(* CODESYS project IOoverNode

Project tree, tasks and I/O mapping:
  Device : XC303, Eaton Automation, version 3.5.16.60
      unmapped channels: Output, Input
    application Application
      libraries: EA_XN300_CAN, 3.5.7.3 (Eaton Automation); Standard, 3.5.15.0 (System); CAA CiA 405, 3.5.15.0 (CAA Technical Workgroup)
      task DatasourcesTask (cyclic, interval 50 ms, priority 31) calls Datasources.Datasources_PRG
      task MainTask (cyclic, interval t#10ms, priority 1) calls PLC_PRG
      function block InputData [ST]
      program PLC_PRG [ST]
      program PRG_PLC [CFC]
    CANbus : CANbus, Eaton Automation, order no. 
      , version 3.5.15.0
        settings: Baudrate = 500 kbit/s
      CANopen_Manager : CANopen_Manager, Eaton Automation, version 3.5.16.0
          settings: CANopen NodeID = 10; ConfigVersion = 50659584
        DA1 : DA1, Eaton Industries, order no. 0, version 3.5.16.100
            settings: General Options.Optional Device = TRUE; NODEIDSAVED = 4; SDO Timeout = 1000000; PDO_Autoconfig = FALSE; EXPERTSETTINGS = True; Emergency-General Parameters.Emergency COBID = 16#00000084; Heartbeat-Producer Time = 200; PDO 16#1400.COBID = 16#40000204; Process by CANopenManager = TRUE; PDO 16#1401.COBID = 16#C0000304; Generic COBID = '$NODEID+16#C0000300'; Process by CANopenManager = TRUE; PDO 16#1800.COBID = 16#40000184; PDO 16#1800.Transmission Type = 16#FF; PDO 16#1800.Event Timer = 0; Process by CANopenManager = TRUE; PDO 16#1801.COBID = 16#C0000284; PDO 16#1801.Event Timer = 0; Generic COBID = '$NODEID+16#C0000280'; Process by CANopenManager = TRUE; Control Command Register.Subindex = 16#00; Speed Reference.Subindex = 16#00; Torque Reference.Subindex = 16#00; User Ramp.Subindex = 16#00; no-name.Index = 16#0006; no-name.Subindex = 16#00; no-name.Index = 16#0006; no-name.Subindex = 16#00; no-name.Index = 16#0006; no-name.Subindex = 16#00; no-name.Index = 16#0006; no-name.Subindex = 16#00; Drive Status Register.Subindex = 16#00; Motor Speed.Subindex = 16#00; Motor Current.Subindex = 16#00; Motor Torque.Subindex = 16#00; Motor Power.Subindex = 16#00; Drive Temperature.Subindex = 16#00; DC Bus Voltage.Subindex = 16#00; Motor Speed (Internal).Subindex = 16#00;
              SDO List.Set COB-ID sync.Index = 16#1005; SDO List.Set COB-ID sync.Subindex = 16#00; SDO List.Set COB-ID sync.Value = 16#00000080; SDO List.Set COB-ID sync.Size = 32; SDO List.Set COB-ID sync.AbortIfError = FALSE; SDO List.Set COB-ID sync.JumpToLine = FALSE; SDO List.Set COB-ID sync.Line = 0; SDO List.Set Guardtime.Index = 16#100C; SDO List.Set Guardtime.Subindex = 16#00; SDO List.Set Guardtime.Value = 16#00000000; SDO List.Set Guardtime.Size = 16; SDO List.Set Guardtime.AbortIfError = FALSE; SDO List.Set Guardtime.JumpToLine = FALSE; SDO List.Set Guardtime.Line = 0; SDO List.Set Lifetime.Index = 16#100D; SDO List.Set Lifetime.Subindex = 16#00; SDO List.Set Lifetime.Value = 16#00000000; SDO List.Set Lifetime.Size = 8; SDO List.Set Lifetime.AbortIfError = FALSE; SDO List.Set Lifetime.JumpToLine = FALSE; SDO List.Set Lifetime.Line = 0; SDO List.Disable Emcy CobID.Index = 16#1014; SDO List.Disable Emcy CobID.Subindex = 16#00; SDO List.Disable Emcy CobID.Value = 16#80000084; SDO List.Disable Emcy CobID.Size = 32; SDO List.Disable Emcy CobID.AbortIfError = FALSE; SDO List.Disable Emcy CobID.JumpToLine = FALSE; SDO List.Disable Emcy CobID.Line = 0; SDO List.Set Emcy CobID.Index = 16#1014; SDO List.Set Emcy CobID.Subindex = 16#00; SDO List.Set Emcy CobID.Value = 16#00000084; SDO List.Set Emcy CobID.Size = 32; SDO List.Set Emcy CobID.AbortIfError = FALSE; SDO List.Set Emcy CobID.JumpToLine = FALSE; SDO List.Set Emcy CobID.Line = 0; SDO List.Set Heartbeat Producer.Index = 16#1017; SDO List.Set Heartbeat Producer.Subindex = 16#00; SDO List.Set Heartbeat Producer.Value = 16#000000C8; SDO List.Set Heartbeat Producer.Size = 16; SDO List.Set Heartbeat Producer.AbortIfError = FALSE;
              SDO List.Set Heartbeat Producer.JumpToLine = FALSE; SDO List.Set Heartbeat Producer.Line = 0; SDO List.Disable PDO.Index = 16#1400; SDO List.Disable PDO.Subindex = 16#01; SDO List.Disable PDO.Value = 16#C0000204; SDO List.Disable PDO.Size = 32; SDO List.Disable PDO.AbortIfError = FALSE; SDO List.Disable PDO.JumpToLine = FALSE; SDO List.Disable PDO.Line = 0; SDO List.Set transmission type.Index = 16#1400; SDO List.Set transmission type.Subindex = 16#02; SDO List.Set transmission type.Value = 16#FE; SDO List.Set transmission type.Size = 8; SDO List.Set transmission type.AbortIfError = FALSE; SDO List.Set transmission type.JumpToLine = FALSE; SDO List.Set transmission type.Line = 0; SDO List.Clear pdo mapping.Index = 16#1600; SDO List.Clear pdo mapping.Subindex = 16#00; SDO List.Clear pdo mapping.Value = 16#0; SDO List.Clear pdo mapping.Size = 8; SDO List.Clear pdo mapping.AbortIfError = FALSE; SDO List.Clear pdo mapping.JumpToLine = FALSE; SDO List.Clear pdo mapping.Line = 0; SDO List.Set Mapping.Index = 16#1600; SDO List.Set Mapping.Subindex = 16#01; SDO List.Set Mapping.Value = 16#20000010; SDO List.Set Mapping.Size = 32; SDO List.Set Mapping.AbortIfError = FALSE; SDO List.Set Mapping.JumpToLine = FALSE; SDO List.Set Mapping.Line = 0; SDO List.Set Mapping.Index = 16#1600; SDO List.Set Mapping.Subindex = 16#02; SDO List.Set Mapping.Value = 16#20010010; SDO List.Set Mapping.Size = 32; SDO List.Set Mapping.AbortIfError = FALSE; SDO List.Set Mapping.JumpToLine = FALSE; SDO List.Set Mapping.Line = 0; SDO List.Set Mapping.Index = 16#1600; SDO List.Set Mapping.Subindex = 16#03; SDO List.Set Mapping.Value = 16#20020010;
              SDO List.Set Mapping.Size = 32; SDO List.Set Mapping.AbortIfError = FALSE; SDO List.Set Mapping.JumpToLine = FALSE; SDO List.Set Mapping.Line = 0; SDO List.Set Mapping.Index = 16#1600; SDO List.Set Mapping.Subindex = 16#04; SDO List.Set Mapping.Value = 16#20030010; SDO List.Set Mapping.Size = 32; SDO List.Set Mapping.AbortIfError = FALSE; SDO List.Set Mapping.JumpToLine = FALSE; SDO List.Set Mapping.Line = 0; SDO List.Set number of mappings.Index = 16#1600; SDO List.Set number of mappings.Subindex = 16#00; SDO List.Set number of mappings.Value = 16#04; SDO List.Set number of mappings.Size = 8; SDO List.Set number of mappings.AbortIfError = FALSE; SDO List.Set number of mappings.JumpToLine = FALSE; SDO List.Set number of mappings.Line = 0; SDO List.Set and enable COB-ID.Index = 16#1400; SDO List.Set and enable COB-ID.Subindex = 16#01; SDO List.Set and enable COB-ID.Value = 16#40000204; SDO List.Set and enable COB-ID.Size = 32; SDO List.Set and enable COB-ID.AbortIfError = FALSE; SDO List.Set and enable COB-ID.JumpToLine = FALSE; SDO List.Set and enable COB-ID.Line = 0; SDO List.Disable PDO.Index = 16#1401; SDO List.Disable PDO.Subindex = 16#01; SDO List.Disable PDO.Value = 16#C0000304; SDO List.Disable PDO.Size = 32; SDO List.Disable PDO.AbortIfError = FALSE; SDO List.Disable PDO.JumpToLine = FALSE; SDO List.Disable PDO.Line = 0; SDO List.Disable PDO.Index = 16#1800; SDO List.Disable PDO.Subindex = 16#01; SDO List.Disable PDO.Value = 16#C0000184; SDO List.Disable PDO.Size = 32; SDO List.Disable PDO.AbortIfError = FALSE; SDO List.Disable PDO.JumpToLine = FALSE; SDO List.Disable PDO.Line = 0; SDO List.Set transmission type.Index = 16#1800;
              SDO List.Set transmission type.Subindex = 16#02; SDO List.Set transmission type.Value = 16#FF; SDO List.Set transmission type.Size = 8; SDO List.Set transmission type.AbortIfError = FALSE; SDO List.Set transmission type.JumpToLine = FALSE; SDO List.Set transmission type.Line = 0; SDO List.Set inhibit time.Index = 16#1800; SDO List.Set inhibit time.Subindex = 16#03; SDO List.Set inhibit time.Value = 16#0000; SDO List.Set inhibit time.Size = 16; SDO List.Set inhibit time.AbortIfError = FALSE; SDO List.Set inhibit time.JumpToLine = FALSE; SDO List.Set inhibit time.Line = 0; SDO List.Clear pdo mapping.Index = 16#1A00; SDO List.Clear pdo mapping.Subindex = 16#00; SDO List.Clear pdo mapping.Value = 16#0; SDO List.Clear pdo mapping.Size = 8; SDO List.Clear pdo mapping.AbortIfError = FALSE; SDO List.Clear pdo mapping.JumpToLine = FALSE; SDO List.Clear pdo mapping.Line = 0; SDO List.Set Mapping.Index = 16#1A00; SDO List.Set Mapping.Subindex = 16#01; SDO List.Set Mapping.Value = 16#200A0010; SDO List.Set Mapping.Size = 32; SDO List.Set Mapping.AbortIfError = FALSE; SDO List.Set Mapping.JumpToLine = FALSE; SDO List.Set Mapping.Line = 0; SDO List.Set Mapping.Index = 16#1A00; SDO List.Set Mapping.Subindex = 16#02; SDO List.Set Mapping.Value = 16#200B0010; SDO List.Set Mapping.Size = 32; SDO List.Set Mapping.AbortIfError = FALSE; SDO List.Set Mapping.JumpToLine = FALSE; SDO List.Set Mapping.Line = 0; SDO List.Set Mapping.Index = 16#1A00; SDO List.Set Mapping.Subindex = 16#03; SDO List.Set Mapping.Value = 16#200D0010; SDO List.Set Mapping.Size = 32; SDO List.Set Mapping.AbortIfError = FALSE; SDO List.Set Mapping.JumpToLine = FALSE;
              SDO List.Set Mapping.Line = 0; SDO List.Set Mapping.Index = 16#1A00; SDO List.Set Mapping.Subindex = 16#04; SDO List.Set Mapping.Value = 16#200E0010; SDO List.Set Mapping.Size = 32; SDO List.Set Mapping.AbortIfError = FALSE; SDO List.Set Mapping.JumpToLine = FALSE; SDO List.Set Mapping.Line = 0; SDO List.Set number of mappings.Index = 16#1A00; SDO List.Set number of mappings.Subindex = 16#00; SDO List.Set number of mappings.Value = 16#04; SDO List.Set number of mappings.Size = 8; SDO List.Set number of mappings.AbortIfError = FALSE; SDO List.Set number of mappings.JumpToLine = FALSE; SDO List.Set number of mappings.Line = 0; SDO List.Set and enable COB-ID.Index = 16#1800; SDO List.Set and enable COB-ID.Subindex = 16#01; SDO List.Set and enable COB-ID.Value = 16#40000184; SDO List.Set and enable COB-ID.Size = 32; SDO List.Set and enable COB-ID.AbortIfError = FALSE; SDO List.Set and enable COB-ID.JumpToLine = FALSE; SDO List.Set and enable COB-ID.Line = 0; SDO List.Disable PDO.Index = 16#1801; SDO List.Disable PDO.Subindex = 16#01; SDO List.Disable PDO.Value = 16#C0000284; SDO List.Disable PDO.Size = 32; SDO List.Disable PDO.AbortIfError = FALSE; SDO List.Disable PDO.JumpToLine = FALSE; SDO List.Disable PDO.Line = 0; ConfigVersion = 50659584
            unmapped channels: Control Command Register, Speed Reference, Torque Reference, User Ramp, Drive Status Register, Motor Speed, Motor Current, Motor Torque
        DC1 : DC1, Eaton, order no. 0, version 3.5.16.100
            settings: General Options.Optional Device = TRUE; NODEIDSAVED = 3; SDO Timeout = 1000000; PDO_Autoconfig = FALSE; EXPERTSETTINGS = True; Emergency-General Parameters.Emergency COBID = 16#00000083; Heartbeat-Producer Time = 200; PDO 16#1400.COBID = 16#40000203; PDO 16#1400.Transmission Type = 16#FE; Process by CANopenManager = TRUE; PDO 16#1401.COBID = 16#C0000303; Generic COBID = '$NODEID+16#C0000300'; Process by CANopenManager = TRUE; PDO 16#1800.COBID = 16#40000183; PDO 16#1800.Event Timer = 0; Process by CANopenManager = TRUE; PDO 16#1801.COBID = 16#C0000283; PDO 16#1801.Event Timer = 0; Generic COBID = '$NODEID+16#C0000280'; Process by CANopenManager = TRUE; Control Command Register.Subindex = 16#00; Speed Reference.Subindex = 16#00; User Ramp.Subindex = 16#00; no-name.Index = 16#0006; no-name.Subindex = 16#00; no-name.Index = 16#0006; no-name.Subindex = 16#00; no-name.Index = 16#0006; no-name.Subindex = 16#00; no-name.Index = 16#0006; no-name.Subindex = 16#00; Drive Status Register.Subindex = 16#00; Motor Speed.Subindex = 16#00; Motor Current.Subindex = 16#00; Drive Temperature.Subindex = 16#00; DC Bus Voltage.Subindex = 16#00; Digital Input Status.Subindex = 16#00; Analog Input 1.Subindex = 16#00; Analog Input 2.Subindex = 16#00; SDO List.Set COB-ID sync.Index = 16#1005;
              SDO List.Set COB-ID sync.Subindex = 16#00; SDO List.Set COB-ID sync.Value = 16#00000080; SDO List.Set COB-ID sync.Size = 32; SDO List.Set COB-ID sync.AbortIfError = FALSE; SDO List.Set COB-ID sync.JumpToLine = FALSE; SDO List.Set COB-ID sync.Line = 0; SDO List.Set Guardtime.Index = 16#100C; SDO List.Set Guardtime.Subindex = 16#00; SDO List.Set Guardtime.Value = 16#00000000; SDO List.Set Guardtime.Size = 16; SDO List.Set Guardtime.AbortIfError = FALSE; SDO List.Set Guardtime.JumpToLine = FALSE; SDO List.Set Guardtime.Line = 0; SDO List.Set Lifetime.Index = 16#100D; SDO List.Set Lifetime.Subindex = 16#00; SDO List.Set Lifetime.Value = 16#00000000; SDO List.Set Lifetime.Size = 8; SDO List.Set Lifetime.AbortIfError = FALSE; SDO List.Set Lifetime.JumpToLine = FALSE; SDO List.Set Lifetime.Line = 0; SDO List.Disable Emcy CobID.Index = 16#1014; SDO List.Disable Emcy CobID.Subindex = 16#00; SDO List.Disable Emcy CobID.Value = 16#80000083; SDO List.Disable Emcy CobID.Size = 32; SDO List.Disable Emcy CobID.AbortIfError = FALSE; SDO List.Disable Emcy CobID.JumpToLine = FALSE; SDO List.Disable Emcy CobID.Line = 0; SDO List.Set Emcy CobID.Index = 16#1014; SDO List.Set Emcy CobID.Subindex = 16#00; SDO List.Set Emcy CobID.Value = 16#00000083; SDO List.Set Emcy CobID.Size = 32; SDO List.Set Emcy CobID.AbortIfError = FALSE; SDO List.Set Emcy CobID.JumpToLine = FALSE; SDO List.Set Emcy CobID.Line = 0; SDO List.Set Heartbeat Producer.Index = 16#1017; SDO List.Set Heartbeat Producer.Subindex = 16#00; SDO List.Set Heartbeat Producer.Value = 16#000000C8; SDO List.Set Heartbeat Producer.Size = 16; SDO List.Set Heartbeat Producer.AbortIfError = FALSE; SDO List.Set Heartbeat Producer.JumpToLine = FALSE;
              SDO List.Set Heartbeat Producer.Line = 0; SDO List.Disable PDO.Index = 16#1400; SDO List.Disable PDO.Subindex = 16#01; SDO List.Disable PDO.Value = 16#C0000203; SDO List.Disable PDO.Size = 32; SDO List.Disable PDO.AbortIfError = FALSE; SDO List.Disable PDO.JumpToLine = FALSE; SDO List.Disable PDO.Line = 0; SDO List.Set transmission type.Index = 16#1400; SDO List.Set transmission type.Subindex = 16#02; SDO List.Set transmission type.Value = 16#FE; SDO List.Set transmission type.Size = 8; SDO List.Set transmission type.AbortIfError = FALSE; SDO List.Set transmission type.JumpToLine = FALSE; SDO List.Set transmission type.Line = 0; SDO List.Clear pdo mapping.Index = 16#1600; SDO List.Clear pdo mapping.Subindex = 16#00; SDO List.Clear pdo mapping.Value = 16#0; SDO List.Clear pdo mapping.Size = 8; SDO List.Clear pdo mapping.AbortIfError = FALSE; SDO List.Clear pdo mapping.JumpToLine = FALSE; SDO List.Clear pdo mapping.Line = 0; SDO List.Set Mapping.Index = 16#1600; SDO List.Set Mapping.Subindex = 16#01; SDO List.Set Mapping.Value = 16#20000010; SDO List.Set Mapping.Size = 32; SDO List.Set Mapping.AbortIfError = FALSE; SDO List.Set Mapping.JumpToLine = FALSE; SDO List.Set Mapping.Line = 0; SDO List.Set Mapping.Index = 16#1600; SDO List.Set Mapping.Subindex = 16#02; SDO List.Set Mapping.Value = 16#20010010; SDO List.Set Mapping.Size = 32; SDO List.Set Mapping.AbortIfError = FALSE; SDO List.Set Mapping.JumpToLine = FALSE; SDO List.Set Mapping.Line = 0; SDO List.Set Mapping.Index = 16#1600; SDO List.Set Mapping.Subindex = 16#03; SDO List.Set Mapping.Value = 16#20030010; SDO List.Set Mapping.Size = 32;
              SDO List.Set Mapping.AbortIfError = FALSE; SDO List.Set Mapping.JumpToLine = FALSE; SDO List.Set Mapping.Line = 0; SDO List.Set number of mappings.Index = 16#1600; SDO List.Set number of mappings.Subindex = 16#00; SDO List.Set number of mappings.Value = 16#03; SDO List.Set number of mappings.Size = 8; SDO List.Set number of mappings.AbortIfError = FALSE; SDO List.Set number of mappings.JumpToLine = FALSE; SDO List.Set number of mappings.Line = 0; SDO List.Set and enable COB-ID.Index = 16#1400; SDO List.Set and enable COB-ID.Subindex = 16#01; SDO List.Set and enable COB-ID.Value = 16#40000203; SDO List.Set and enable COB-ID.Size = 32; SDO List.Set and enable COB-ID.AbortIfError = FALSE; SDO List.Set and enable COB-ID.JumpToLine = FALSE; SDO List.Set and enable COB-ID.Line = 0; SDO List.Disable PDO.Index = 16#1401; SDO List.Disable PDO.Subindex = 16#01; SDO List.Disable PDO.Value = 16#C0000303; SDO List.Disable PDO.Size = 32; SDO List.Disable PDO.AbortIfError = FALSE; SDO List.Disable PDO.JumpToLine = FALSE; SDO List.Disable PDO.Line = 0; SDO List.Disable PDO.Index = 16#1800; SDO List.Disable PDO.Subindex = 16#01; SDO List.Disable PDO.Value = 16#C0000183; SDO List.Disable PDO.Size = 32; SDO List.Disable PDO.AbortIfError = FALSE; SDO List.Disable PDO.JumpToLine = FALSE; SDO List.Disable PDO.Line = 0; SDO List.Set transmission type.Index = 16#1800; SDO List.Set transmission type.Subindex = 16#02; SDO List.Set transmission type.Value = 16#FF; SDO List.Set transmission type.Size = 8; SDO List.Set transmission type.AbortIfError = FALSE; SDO List.Set transmission type.JumpToLine = FALSE; SDO List.Set transmission type.Line = 0; SDO List.Set inhibit time.Index = 16#1800; SDO List.Set inhibit time.Subindex = 16#03;
              SDO List.Set inhibit time.Value = 16#0000; SDO List.Set inhibit time.Size = 16; SDO List.Set inhibit time.AbortIfError = FALSE; SDO List.Set inhibit time.JumpToLine = FALSE; SDO List.Set inhibit time.Line = 0; SDO List.Clear pdo mapping.Index = 16#1A00; SDO List.Clear pdo mapping.Subindex = 16#00; SDO List.Clear pdo mapping.Value = 16#0; SDO List.Clear pdo mapping.Size = 8; SDO List.Clear pdo mapping.AbortIfError = FALSE; SDO List.Clear pdo mapping.JumpToLine = FALSE; SDO List.Clear pdo mapping.Line = 0; SDO List.Set Mapping.Index = 16#1A00; SDO List.Set Mapping.Subindex = 16#01; SDO List.Set Mapping.Value = 16#200A0010; SDO List.Set Mapping.Size = 32; SDO List.Set Mapping.AbortIfError = FALSE; SDO List.Set Mapping.JumpToLine = FALSE; SDO List.Set Mapping.Line = 0; SDO List.Set Mapping.Index = 16#1A00; SDO List.Set Mapping.Subindex = 16#02; SDO List.Set Mapping.Value = 16#200B0010; SDO List.Set Mapping.Size = 32; SDO List.Set Mapping.AbortIfError = FALSE; SDO List.Set Mapping.JumpToLine = FALSE; SDO List.Set Mapping.Line = 0; SDO List.Set Mapping.Index = 16#1A00; SDO List.Set Mapping.Subindex = 16#03; SDO List.Set Mapping.Value = 16#200D0010; SDO List.Set Mapping.Size = 32; SDO List.Set Mapping.AbortIfError = FALSE; SDO List.Set Mapping.JumpToLine = FALSE; SDO List.Set Mapping.Line = 0; SDO List.Set Mapping.Index = 16#1A00; SDO List.Set Mapping.Subindex = 16#04; SDO List.Set Mapping.Value = 16#20100010; SDO List.Set Mapping.Size = 32; SDO List.Set Mapping.AbortIfError = FALSE; SDO List.Set Mapping.JumpToLine = FALSE; SDO List.Set Mapping.Line = 0;
              SDO List.Set number of mappings.Index = 16#1A00; SDO List.Set number of mappings.Subindex = 16#00; SDO List.Set number of mappings.Value = 16#04; SDO List.Set number of mappings.Size = 8; SDO List.Set number of mappings.AbortIfError = FALSE; SDO List.Set number of mappings.JumpToLine = FALSE; SDO List.Set number of mappings.Line = 0; SDO List.Set and enable COB-ID.Index = 16#1800; SDO List.Set and enable COB-ID.Subindex = 16#01; SDO List.Set and enable COB-ID.Value = 16#40000183; SDO List.Set and enable COB-ID.Size = 32; SDO List.Set and enable COB-ID.AbortIfError = FALSE; SDO List.Set and enable COB-ID.JumpToLine = FALSE; SDO List.Set and enable COB-ID.Line = 0; SDO List.Disable PDO.Index = 16#1801; SDO List.Disable PDO.Subindex = 16#01; SDO List.Disable PDO.Value = 16#C0000283; SDO List.Disable PDO.Size = 32; SDO List.Disable PDO.AbortIfError = FALSE; SDO List.Disable PDO.JumpToLine = FALSE; SDO List.Disable PDO.Line = 0; ConfigVersion = 50659584
            unmapped channels: Control Command Register, Speed Reference, User Ramp, Drive Status Register, Motor Speed, Motor Current, Drive Temperature
        XN_312_GW_CAN : XN-312-GW-CAN, Eaton Automation, order no. 178782, version Revision=16#00000000, FileVersion=1.5
            settings: NODEIDSAVED = 2; SDO Timeout = 1000000; EXPERTSETTINGS = FALSE; Nodeguarding.Guard Time = 0 ms; Nodeguarding.Life Time Factor = 0; Emergency-General Parameters.Emergency COBID = 16#00000082; Heartbeat-Producer Time = 200; Settings.COBID = 16#00000202; Settings.Transmission Type = 16#FF; Settings.available PDO-Parameter.Inhibit Time available = FALSE; Settings.available PDO-Parameter.Event Timer available = FALSE; Settings.Inhibit Time = 0; Settings.Event Timer = 0; Generic COBID = '$NODEID+16#0200'; Process by CANopenManager = TRUE; Settings.COBID = 16#00000302; Settings.Transmission Type = 16#FF; Settings.available PDO-Parameter.Inhibit Time available = FALSE; Settings.available PDO-Parameter.Event Timer available = FALSE; Settings.Inhibit Time = 0; Settings.Event Timer = 0; Generic COBID = '$NODEID+16#0300'; Process by CANopenManager = TRUE; Settings.COBID = 16#00000182; Settings.Transmission Type = 16#FF; Settings.available PDO-Parameter.Inhibit Time available = TRUE; Settings.available PDO-Parameter.Event Timer available = TRUE; Settings.Inhibit Time = 0; Settings.Event Timer = 0; Generic COBID = '$NODEID+16#0180'; Process by CANopenManager = TRUE; Settings.COBID = 16#00000282; Settings.Transmission Type = 16#FF; Settings.available PDO-Parameter.Inhibit Time available = TRUE; Settings.available PDO-Parameter.Event Timer available = TRUE; Settings.Inhibit Time = 0; Settings.Event Timer = 0; Generic COBID = '$NODEID+16#0280'; Process by CANopenManager = TRUE; Heartbeat-Consuming1.Heartbeat-Time = 300 ms;
              Q-Byte : XN_322_16DIO_PD05_1.Index = 16#6200; Q-Byte : XN_322_16DIO_PD05_1.Subindex = 16#01; Q-Byte : XN_322_16DIO_PD05_1.ObjectLength = 8; Q-Byte : XN_322_4DO_RNO.Index = 16#6200; Q-Byte : XN_322_4DO_RNO.Subindex = 16#02; Q-Byte : XN_322_4DO_RNO.ObjectLength = 8; Q-WORD : XN_322_4AIO_U2.Index = 16#6411; Q-WORD : XN_322_4AIO_U2.Subindex = 16#01; Q-WORD : XN_322_4AIO_U2.ObjectLength = 16; Q-WORD : XN_322_4AIO_U2.Index = 16#6411; Q-WORD : XN_322_4AIO_U2.Subindex = 16#02; Q-WORD : XN_322_4AIO_U2.ObjectLength = 16; I-Byte : XN_322_16DIO_PD05_1.Index = 16#6000; I-Byte : XN_322_16DIO_PD05_1.Subindex = 16#01; I-Byte : XN_322_16DIO_PD05_1.ObjectLength = 8; I-WORD : XN_322_4AIO_U2.Index = 16#6401; I-WORD : XN_322_4AIO_U2.Subindex = 16#01; I-WORD : XN_322_4AIO_U2.ObjectLength = 16; I-WORD : XN_322_4AIO_U2.Index = 16#6401; I-WORD : XN_322_4AIO_U2.Subindex = 16#02; I-WORD : XN_322_4AIO_U2.ObjectLength = 16; SDO List.Set COB-ID sync.Index = 16#1005; SDO List.Set COB-ID sync.Subindex = 16#00; SDO List.Set COB-ID sync.Value = 16#00000080; SDO List.Set COB-ID sync.Size = 32; SDO List.Set COB-ID sync.AbortIfError = FALSE; SDO List.Set COB-ID sync.JumpToLine = FALSE; SDO List.Set COB-ID sync.Line = 0; SDO List.Set Guardtime.Index = 16#100C; SDO List.Set Guardtime.Subindex = 16#00; SDO List.Set Guardtime.Value = 16#00000000; SDO List.Set Guardtime.Size = 16; SDO List.Set Guardtime.AbortIfError = FALSE; SDO List.Set Guardtime.JumpToLine = FALSE; SDO List.Set Guardtime.Line = 0; SDO List.Set Lifetime.Index = 16#100D; SDO List.Set Lifetime.Subindex = 16#00; SDO List.Set Lifetime.Value = 16#00000000; SDO List.Set Lifetime.Size = 8; SDO List.Set Lifetime.AbortIfError = FALSE;
              SDO List.Set Lifetime.JumpToLine = FALSE; SDO List.Set Lifetime.Line = 0; SDO List.Disable Emcy CobID.Index = 16#1014; SDO List.Disable Emcy CobID.Subindex = 16#00; SDO List.Disable Emcy CobID.Value = 16#80000082; SDO List.Disable Emcy CobID.Size = 32; SDO List.Disable Emcy CobID.AbortIfError = FALSE; SDO List.Disable Emcy CobID.JumpToLine = FALSE; SDO List.Disable Emcy CobID.Line = 0; SDO List.Set Emcy CobID.Index = 16#1014; SDO List.Set Emcy CobID.Subindex = 16#00; SDO List.Set Emcy CobID.Value = 16#00000082; SDO List.Set Emcy CobID.Size = 32; SDO List.Set Emcy CobID.AbortIfError = FALSE; SDO List.Set Emcy CobID.JumpToLine = FALSE; SDO List.Set Emcy CobID.Line = 0; SDO List.Set Heartbeat Consumer.Index = 16#1016; SDO List.Set Heartbeat Consumer.Subindex = 16#01; SDO List.Set Heartbeat Consumer.Value = 16#0001012C; SDO List.Set Heartbeat Consumer.Size = 32; SDO List.Set Heartbeat Consumer.AbortIfError = FALSE; SDO List.Set Heartbeat Consumer.JumpToLine = FALSE; SDO List.Set Heartbeat Consumer.Line = 0; SDO List.Set Heartbeat Consumer.Index = 16#1016; SDO List.Set Heartbeat Consumer.Subindex = 16#02; SDO List.Set Heartbeat Consumer.Value = 0; SDO List.Set Heartbeat Consumer.Size = 32; SDO List.Set Heartbeat Consumer.AbortIfError = FALSE; SDO List.Set Heartbeat Consumer.JumpToLine = FALSE; SDO List.Set Heartbeat Consumer.Line = 0; SDO List.Set Heartbeat Consumer.Index = 16#1016; SDO List.Set Heartbeat Consumer.Subindex = 16#03; SDO List.Set Heartbeat Consumer.Value = 0; SDO List.Set Heartbeat Consumer.Size = 32; SDO List.Set Heartbeat Consumer.AbortIfError = FALSE; SDO List.Set Heartbeat Consumer.JumpToLine = FALSE; SDO List.Set Heartbeat Consumer.Line = 0; SDO List.Set Heartbeat Consumer.Index = 16#1016; SDO List.Set Heartbeat Consumer.Subindex = 16#04; SDO List.Set Heartbeat Consumer.Value = 0;
              SDO List.Set Heartbeat Consumer.Size = 32; SDO List.Set Heartbeat Consumer.AbortIfError = FALSE; SDO List.Set Heartbeat Consumer.JumpToLine = FALSE; SDO List.Set Heartbeat Consumer.Line = 0; SDO List.Set Heartbeat Producer.Index = 16#1017; SDO List.Set Heartbeat Producer.Subindex = 16#00; SDO List.Set Heartbeat Producer.Value = 16#000000C8; SDO List.Set Heartbeat Producer.Size = 16; SDO List.Set Heartbeat Producer.AbortIfError = FALSE; SDO List.Set Heartbeat Producer.JumpToLine = FALSE; SDO List.Set Heartbeat Producer.Line = 0; SDO List.Disable PDO.Index = 16#1400; SDO List.Disable PDO.Subindex = 16#01; SDO List.Disable PDO.Value = 16#80000202; SDO List.Disable PDO.Size = 32; SDO List.Disable PDO.AbortIfError = FALSE; SDO List.Disable PDO.JumpToLine = FALSE; SDO List.Disable PDO.Line = 0; SDO List.Set transmission type.Index = 16#1400; SDO List.Set transmission type.Subindex = 16#02; SDO List.Set transmission type.Value = 16#FF; SDO List.Set transmission type.Size = 8; SDO List.Set transmission type.AbortIfError = FALSE; SDO List.Set transmission type.JumpToLine = FALSE; SDO List.Set transmission type.Line = 0; SDO List.Clear pdo mapping.Index = 16#1600; SDO List.Clear pdo mapping.Subindex = 16#00; SDO List.Clear pdo mapping.Value = 16#0; SDO List.Clear pdo mapping.Size = 8; SDO List.Clear pdo mapping.AbortIfError = FALSE; SDO List.Clear pdo mapping.JumpToLine = FALSE; SDO List.Clear pdo mapping.Line = 0; SDO List.Set Mapping.Index = 16#1600; SDO List.Set Mapping.Subindex = 16#01; SDO List.Set Mapping.Value = 16#62000108; SDO List.Set Mapping.Size = 32; SDO List.Set Mapping.AbortIfError = FALSE; SDO List.Set Mapping.JumpToLine = FALSE; SDO List.Set Mapping.Line = 0; SDO List.Set Mapping.Index = 16#1600;
              SDO List.Set Mapping.Subindex = 16#02; SDO List.Set Mapping.Value = 16#62000208; SDO List.Set Mapping.Size = 32; SDO List.Set Mapping.AbortIfError = FALSE; SDO List.Set Mapping.JumpToLine = FALSE; SDO List.Set Mapping.Line = 0; SDO List.Set number of mappings.Index = 16#1600; SDO List.Set number of mappings.Subindex = 16#00; SDO List.Set number of mappings.Value = 16#02; SDO List.Set number of mappings.Size = 8; SDO List.Set number of mappings.AbortIfError = FALSE; SDO List.Set number of mappings.JumpToLine = FALSE; SDO List.Set number of mappings.Line = 0; SDO List.Set and enable COB-ID.Index = 16#1400; SDO List.Set and enable COB-ID.Subindex = 16#01; SDO List.Set and enable COB-ID.Value = 16#00000202; SDO List.Set and enable COB-ID.Size = 32; SDO List.Set and enable COB-ID.AbortIfError = FALSE; SDO List.Set and enable COB-ID.JumpToLine = FALSE; SDO List.Set and enable COB-ID.Line = 0; SDO List.Disable PDO.Index = 16#1401; SDO List.Disable PDO.Subindex = 16#01; SDO List.Disable PDO.Value = 16#80000302; SDO List.Disable PDO.Size = 32; SDO List.Disable PDO.AbortIfError = FALSE; SDO List.Disable PDO.JumpToLine = FALSE; SDO List.Disable PDO.Line = 0; SDO List.Set transmission type.Index = 16#1401; SDO List.Set transmission type.Subindex = 16#02; SDO List.Set transmission type.Value = 16#FF; SDO List.Set transmission type.Size = 8; SDO List.Set transmission type.AbortIfError = FALSE; SDO List.Set transmission type.JumpToLine = FALSE; SDO List.Set transmission type.Line = 0; SDO List.Clear pdo mapping.Index = 16#1601; SDO List.Clear pdo mapping.Subindex = 16#00; SDO List.Clear pdo mapping.Value = 16#0; SDO List.Clear pdo mapping.Size = 8; SDO List.Clear pdo mapping.AbortIfError = FALSE; SDO List.Clear pdo mapping.JumpToLine = FALSE;
              SDO List.Clear pdo mapping.Line = 0; SDO List.Set Mapping.Index = 16#1601; SDO List.Set Mapping.Subindex = 16#01; SDO List.Set Mapping.Value = 16#64110110; SDO List.Set Mapping.Size = 32; SDO List.Set Mapping.AbortIfError = FALSE; SDO List.Set Mapping.JumpToLine = FALSE; SDO List.Set Mapping.Line = 0; SDO List.Set Mapping.Index = 16#1601; SDO List.Set Mapping.Subindex = 16#02; SDO List.Set Mapping.Value = 16#64110210; SDO List.Set Mapping.Size = 32; SDO List.Set Mapping.AbortIfError = FALSE; SDO List.Set Mapping.JumpToLine = FALSE; SDO List.Set Mapping.Line = 0; SDO List.Set number of mappings.Index = 16#1601; SDO List.Set number of mappings.Subindex = 16#00; SDO List.Set number of mappings.Value = 16#02; SDO List.Set number of mappings.Size = 8; SDO List.Set number of mappings.AbortIfError = FALSE; SDO List.Set number of mappings.JumpToLine = FALSE; SDO List.Set number of mappings.Line = 0; SDO List.Set and enable COB-ID.Index = 16#1401; SDO List.Set and enable COB-ID.Subindex = 16#01; SDO List.Set and enable COB-ID.Value = 16#00000302; SDO List.Set and enable COB-ID.Size = 32; SDO List.Set and enable COB-ID.AbortIfError = FALSE; SDO List.Set and enable COB-ID.JumpToLine = FALSE; SDO List.Set and enable COB-ID.Line = 0; SDO List.Disable PDO.Index = 16#1800; SDO List.Disable PDO.Subindex = 16#01; SDO List.Disable PDO.Value = 16#80000182; SDO List.Disable PDO.Size = 32; SDO List.Disable PDO.AbortIfError = FALSE; SDO List.Disable PDO.JumpToLine = FALSE; SDO List.Disable PDO.Line = 0; SDO List.Set transmission type.Index = 16#1800; SDO List.Set transmission type.Subindex = 16#02; SDO List.Set transmission type.Value = 16#FF; SDO List.Set transmission type.Size = 8;
              SDO List.Set transmission type.AbortIfError = FALSE; SDO List.Set transmission type.JumpToLine = FALSE; SDO List.Set transmission type.Line = 0; SDO List.Set inhibit time.Index = 16#1800; SDO List.Set inhibit time.Subindex = 16#03; SDO List.Set inhibit time.Value = 16#0000; SDO List.Set inhibit time.Size = 16; SDO List.Set inhibit time.AbortIfError = FALSE; SDO List.Set inhibit time.JumpToLine = FALSE; SDO List.Set inhibit time.Line = 0; SDO List.Set event time.Index = 16#1800; SDO List.Set event time.Subindex = 16#05; SDO List.Set event time.Value = 16#0000; SDO List.Set event time.Size = 16; SDO List.Set event time.AbortIfError = FALSE; SDO List.Set event time.JumpToLine = FALSE; SDO List.Set event time.Line = 0; SDO List.Clear pdo mapping.Index = 16#1A00; SDO List.Clear pdo mapping.Subindex = 16#00; SDO List.Clear pdo mapping.Value = 16#0; SDO List.Clear pdo mapping.Size = 8; SDO List.Clear pdo mapping.AbortIfError = FALSE; SDO List.Clear pdo mapping.JumpToLine = FALSE; SDO List.Clear pdo mapping.Line = 0; SDO List.Set Mapping.Index = 16#1A00; SDO List.Set Mapping.Subindex = 16#01; SDO List.Set Mapping.Value = 16#60000108; SDO List.Set Mapping.Size = 32; SDO List.Set Mapping.AbortIfError = FALSE; SDO List.Set Mapping.JumpToLine = FALSE; SDO List.Set Mapping.Line = 0; SDO List.Set number of mappings.Index = 16#1A00; SDO List.Set number of mappings.Subindex = 16#00; SDO List.Set number of mappings.Value = 16#01; SDO List.Set number of mappings.Size = 8; SDO List.Set number of mappings.AbortIfError = FALSE; SDO List.Set number of mappings.JumpToLine = FALSE; SDO List.Set number of mappings.Line = 0; SDO List.Set and enable COB-ID.Index = 16#1800; SDO List.Set and enable COB-ID.Subindex = 16#01;
              SDO List.Set and enable COB-ID.Value = 16#00000182; SDO List.Set and enable COB-ID.Size = 32; SDO List.Set and enable COB-ID.AbortIfError = FALSE; SDO List.Set and enable COB-ID.JumpToLine = FALSE; SDO List.Set and enable COB-ID.Line = 0; SDO List.Disable PDO.Index = 16#1801; SDO List.Disable PDO.Subindex = 16#01; SDO List.Disable PDO.Value = 16#80000282; SDO List.Disable PDO.Size = 32; SDO List.Disable PDO.AbortIfError = FALSE; SDO List.Disable PDO.JumpToLine = FALSE; SDO List.Disable PDO.Line = 0; SDO List.Set transmission type.Index = 16#1801; SDO List.Set transmission type.Subindex = 16#02; SDO List.Set transmission type.Value = 16#FF; SDO List.Set transmission type.Size = 8; SDO List.Set transmission type.AbortIfError = FALSE; SDO List.Set transmission type.JumpToLine = FALSE; SDO List.Set transmission type.Line = 0; SDO List.Set inhibit time.Index = 16#1801; SDO List.Set inhibit time.Subindex = 16#03; SDO List.Set inhibit time.Value = 16#0000; SDO List.Set inhibit time.Size = 16; SDO List.Set inhibit time.AbortIfError = FALSE; SDO List.Set inhibit time.JumpToLine = FALSE; SDO List.Set inhibit time.Line = 0; SDO List.Set event time.Index = 16#1801; SDO List.Set event time.Subindex = 16#05; SDO List.Set event time.Value = 16#0000; SDO List.Set event time.Size = 16; SDO List.Set event time.AbortIfError = FALSE; SDO List.Set event time.JumpToLine = FALSE; SDO List.Set event time.Line = 0; SDO List.Clear pdo mapping.Index = 16#1A01; SDO List.Clear pdo mapping.Subindex = 16#00; SDO List.Clear pdo mapping.Value = 16#0; SDO List.Clear pdo mapping.Size = 8; SDO List.Clear pdo mapping.AbortIfError = FALSE; SDO List.Clear pdo mapping.JumpToLine = FALSE; SDO List.Clear pdo mapping.Line = 0;
              SDO List.Set Mapping.Index = 16#1A01; SDO List.Set Mapping.Subindex = 16#01; SDO List.Set Mapping.Value = 16#64010110; SDO List.Set Mapping.Size = 32; SDO List.Set Mapping.AbortIfError = FALSE; SDO List.Set Mapping.JumpToLine = FALSE; SDO List.Set Mapping.Line = 0; SDO List.Set Mapping.Index = 16#1A01; SDO List.Set Mapping.Subindex = 16#02; SDO List.Set Mapping.Value = 16#64010210; SDO List.Set Mapping.Size = 32; SDO List.Set Mapping.AbortIfError = FALSE; SDO List.Set Mapping.JumpToLine = FALSE; SDO List.Set Mapping.Line = 0; SDO List.Set number of mappings.Index = 16#1A01; SDO List.Set number of mappings.Subindex = 16#00; SDO List.Set number of mappings.Value = 16#02; SDO List.Set number of mappings.Size = 8; SDO List.Set number of mappings.AbortIfError = FALSE; SDO List.Set number of mappings.JumpToLine = FALSE; SDO List.Set number of mappings.Line = 0; SDO List.Set and enable COB-ID.Index = 16#1801; SDO List.Set and enable COB-ID.Subindex = 16#01; SDO List.Set and enable COB-ID.Value = 16#00000282; SDO List.Set and enable COB-ID.Size = 32; SDO List.Set and enable COB-ID.AbortIfError = FALSE; SDO List.Set and enable COB-ID.JumpToLine = FALSE; SDO List.Set and enable COB-ID.Line = 0; ConfigVersion = 50659584
          XN_322_16DIO_PD05_1 : XN-322-16DIO-PD05, Eaton Automation, order no. 0, version Revision=16#00000000, FileVersion=1.5
              settings: Number of Params = 1; Q-Byte : XN_322_16DIO_PD05_1.Index = 16#6200; Q-Byte : XN_322_16DIO_PD05_1.Subindex = 16#01; Q-Byte : XN_322_16DIO_PD05_1.Startbit = 0; Q-Byte : XN_322_16DIO_PD05_1.Endbit = 7; Number of Params = 1; I-Byte : XN_322_16DIO_PD05_1.Index = 16#6000; I-Byte : XN_322_16DIO_PD05_1.Subindex = 16#01; I-Byte : XN_322_16DIO_PD05_1.Startbit = 0; I-Byte : XN_322_16DIO_PD05_1.Endbit = 7
              unmapped channels: Q-Byte : XN_322_16DIO_PD05_1, I-Byte : XN_322_16DIO_PD05_1
          XN_322_4AIO_U2 : XN-322-4AIO-U2, Eaton Automation, order no. 0, version Revision=16#00000000, FileVersion=1.5
              settings: Number of Params = 2; Q-WORD : XN_322_4AIO_U2.Index = 16#6411; Q-WORD : XN_322_4AIO_U2.Subindex = 16#01; Q-WORD : XN_322_4AIO_U2.Startbit = 0; Q-WORD : XN_322_4AIO_U2.Endbit = 15; Q-WORD : XN_322_4AIO_U2.Index = 16#6411; Q-WORD : XN_322_4AIO_U2.Subindex = 16#02; Q-WORD : XN_322_4AIO_U2.Startbit = 0; Q-WORD : XN_322_4AIO_U2.Endbit = 15; Number of Params = 2; I-WORD : XN_322_4AIO_U2.Index = 16#6401; I-WORD : XN_322_4AIO_U2.Subindex = 16#01; I-WORD : XN_322_4AIO_U2.Startbit = 0; I-WORD : XN_322_4AIO_U2.Endbit = 15; I-WORD : XN_322_4AIO_U2.Index = 16#6401; I-WORD : XN_322_4AIO_U2.Subindex = 16#02; I-WORD : XN_322_4AIO_U2.Startbit = 0; I-WORD : XN_322_4AIO_U2.Endbit = 15
              unmapped channels: Q-WORD : XN_322_4AIO_U2, Q-WORD : XN_322_4AIO_U2, I-WORD : XN_322_4AIO_U2, I-WORD : XN_322_4AIO_U2
          XN_322_4DO_RNO : XN-322-4DO-RNO, Eaton Automation, order no. 0, version Revision=16#00000000, FileVersion=1.5
              settings: Number of Params = 1; Q-Byte : XN_322_4DO_RNO.Index = 16#6200; Q-Byte : XN_322_4DO_RNO.Subindex = 16#02; Q-Byte : XN_322_4DO_RNO.Startbit = 0; Q-Byte : XN_322_4DO_RNO.Endbit = 7
              unmapped channels: Q-Byte : XN_322_4DO_RNO
    Modbus_COM_Port : Modbus COM Port, 3S - Smart Software Solutions GmbH, version 3.5.16.0
        settings: DataBits = 8; StopBits = 1; ComPort = 1
      Modbus_Master_COM_Port : Modbus Master, COM Port, 3S - Smart Software Solutions GmbH, version 3.5.16.0
          settings: Transmission = 'RTU'; ResponseTimeout = 1000; TimeBetweenFrames = 10; Auto-restart communication = TRUE
        Modbus_Slave_DA1 : Modbus Slave, DA1, Eaton Industries, version 3.5.16.100
            settings: SlaveAddress = 4; ResponseTimeout = 1000; UseExtendedFunctionCodes = TRUE
            unmapped channels: ControlCommand, SpeedRef, TorqueReference, ProcessValues
        Modbus_Slave_DC1 : Modbus Slave, DC1, Eaton Industries, version 3.5.16.100
            settings: SlaveAddress = 3; ResponseTimeout = 1000; UseExtendedFunctionCodes = TRUE
            unmapped channels: ControlCommand, SpeedRef, ProcessValues
  XV300 : XV300, Eaton Automation, version 3.5.16.60
    application Application
      libraries: Standard, 3.5.15.0 (System); EA_XN300_CAN, 3.5.7.2 (Eaton Automation)
      task MainTask (cyclic, interval t#10ms, priority 1) calls PLC_PRG
      program PLC_PRG [ST]
    SWD_Master : SWD-Master, Eaton Automation, version 3.5.8.0
      M22_SWD_INC_Profile_2 : M22-SWD-INC Profile 2, Eaton Industries GmbH, order no. 0815, version 3.5.3.0
          unmapped channels: Output 0, Input0, Input1
      M22_SWD_K11LED_B : M22-SWD-K11LED-B, Eaton Industries GmbH, order no. 0815, version 3.5.2.0
          unmapped channels: Output, Input
      M22_SWD_K11LED_W_1 : M22-SWD-K11LED-W, Eaton Industries GmbH, order no. 0815, version 3.5.2.0
          unmapped channels: Output, Input
      M22_SWD_K11LED_W : M22-SWD-K11LED-W, Eaton Industries GmbH, order no. 0815, version 3.5.2.0
          unmapped channels: Output, Input
      M22_SWD_K22LED_R : M22-SWD-K22LED-R, Eaton Industries GmbH, order no. 0815, version 3.5.2.0
          unmapped channels: Output, Input
      M22_SWD_K22LED_W_1 : M22-SWD-K22LED-W, Eaton Industries GmbH, order no. 0815, version 3.5.2.0
          unmapped channels: Output, Input
      M22_SWD_K22LED_W : M22-SWD-K22LED-W, Eaton Industries GmbH, order no. 0815, version 3.5.2.0
          unmapped channels: Output, Input
      M22_SWD_R_Profile_2_1 : M22-SWD-R Profile 2, Eaton Industries GmbH, order no. 0815, version 3.5.2.0
          unmapped channels: Input0, Input1
      M22_SWD_R_Profile_2 : M22-SWD-R Profile 2, Eaton Industries GmbH, order no. 0815, version 3.5.2.0
          unmapped channels: Input0, Input1
      MainMotor : PKE-SWD-32 Profile 3, Eaton Industries GmbH, order no. 0815, version 3.5.16.100
          unmapped channels: Output0, Input0
  libraries: Common Behaviour Model, 3.5.17.0 (3S - Smart Software Solutions GmbH); CAA CiA 405, 3.5.17.0 (CAA Technical Workgroup); BASIC, 3.3.4.0 (OSCAT); Standard, * (System); EA_SWD, 3.5.8.0 (Eaton Automation)
  Basic/
    Enums/
      Error/
        data type teErrorCodeEaton
      PKE/
        data type teCurrentUnit
        data type tePkeErrorCode
        data type teSwitchPos_1_0_A
        data type teTripBlock
        data type teTripReason
      data type teFieldbus
      data type teProtTypecode
      data type teStartTypecode
    FB/
      function block FB_Basic [ST]: FB_Init, GetName, GetPath
      function block FB_BasicWithBehaviour [ST]: GetModelState, ControlCleanupAction, ControlCyclicAction, ControlExitAction, ControlResetAction, ControlStartAction, CleanupAction, CyclicAction, ExitAction, ResetAction, StartAction, IBehaviourModel
      function block FB_HWDeviceBasic [ST]: CyclicAction, eFieldbus, ExitAction, FB_INIT, StartAction
    Interface/
      interface I_HWDevice
      interface IBasicBehaviour: GetModelState, IBehaviourModel
      interface IBasicElement: GetName, GetPath
  FunctionBlock/
    function block FB_Drive [ST]: ACT_MapIO, CyclicAction, Direction, ErrorCode, ExitAction, Fault, FixedFrequency, FreeRunDown, GetParameter, HardwareEnable, ModulName, Operation, QuickStop, rAcceleration, rCurrent, rDeceleration, rEnergy, rVelocity, SetpointReached, SpeedControl, StartAction, TypeCode, ZeroSpeed
    function block FB_ErrorHandler [ST]: AttachDevice, DetachDevice
    function block FB_PKE [ST]: ACKR, ACT_MapModbus, ACT_MapSWD, Class, Contactor, Current_A, CyclicAction, ErrorCode, M_Current, ModulName, ModulPresent, P_xConnected, P_xError, PartTripBlock, PkeStatus, SelectValueIr, StartAction, SwitchState_1_0_A, ThermalMotorImage, TripReason, ZmrAutoHand
  Global Variables/
    global variables GVL_Const
    global variables GVL_ErrorCodeDefEaton
  Interface/
    interface I_ErroHandlerSubject: AttachDevice, DetachDevice
    interface ITF_Base_MotorProtection: Current_A, P_xConnected, P_xError
    interface ITF_Base_MotorStarter: Direction, ErrorCode, Operation
    interface ITF_DIL: Contactor, SwitchState_1_0_A
    interface ITF_Drive: eFieldbus, Fault, FixedFrequency, FreeRunDown, GetParameter, HardwareEnable, ModulName, QuickStop, rAcceleration, rCurrent, rDeceleration, rEnergy, rVelocity, SetpointReached, SpeedControl, TypeCode, ZeroSpeed
    interface ITF_PKE: ACKR, Class, Contactor, Current_A, eFieldbus, ErrorCode, M_Current, ModulName, ModulPresent, PartTripBlock, PkeStatus, SelectValueIr, SwitchState_1_0_A, ThermalMotorImage, TripReason, ZmrAutoHand
  Structs/
    DA1/
      data type teDriveError
      data type teDriveParameter
      data type teDriveTyp
      data type tsCommandAndControl16bit
      data type tsDriveCommandAndSpeed
      data type tsDriveStatusAndSpeed
      data type tsStatusAndFaults16bit
    SWD/
      data type tePkeProfile
      data type tsIB0_PKE_SWD_32
      data type tsIB1_PKE_SWD_32
      data type tsIB4_PKE_SWD_32
      data type tsIB_DIL_SWD_32
      data type tsPKE_ModXTUA
      data type tsPKE_Profil1
      data type tsPKE_Profil2
      data type tsPKE_Profil3
      data type tsQB_DIL_SWD_32
      data type tsQB_PKE_Mod
      data type tsQB_PKE_SWD_32
    data type ts3rdPartyDevicInfo
    data type tsCBMLInfo
    data type tsCmsInterface
    data type tsProtectionDevicInfo
    data type tsStarterDevicInfo
*)

// Structs/ts3rdPartyDevicInfo
(*Device Managment Information from the Part "3rd party" 
	e.g. Motor, Incoder, Temperature Sensor *)
TYPE ts3rdPartyDevicInfo :
STRUCT	
	str3rdTypeCode			: STRING[20]; 		// text string specifiying device 	
	str3rdSupplier			: STRING; 			// Supplier Name					
	str3rdOrderNumber		: STRING[20]; 		// OrderNumber from Supplier		
	str3rdProductionDate	: STRING[20];  		// Producation Date from Device		
	str3rdFirmwareVer		: STRING[20];		// Firmware Version from Device		
	str3rdSerialNum			: STRING[20]; 		// Serial Number from Device		
END_STRUCT
END_TYPE

// Structs/tsCBMLInfo
TYPE tsCBMLInfo :
STRUCT
	xCommit		: BOOL; 
	xDone		: BOOL; 
	xBusy		: BOOL; 
	xError		: BOOL; 
	xAborted	: BOOL; 
	iErrorID	: INT; 
	eState		: CBML.STATE;
	strName		: STRING;
END_STRUCT
END_TYPE

// Structs/tsCmsInterface
//CMS Interface Definition of the Tags between PLC and Gateway
TYPE tsCmsInterface :
STRUCT
	(* Interface Definition Version; between PLC - Gateway - Cloud for CMS *)
	wVersion 				: WORD; 			// the interface version; 			"version":{"value":1.0}	
	(* Position Value of the physikal Device*)
	rPosLat					: REAL; 			// latitude of Geo positions 		"posLat":{"value":<POS_LAT>}
	rPosLon					: REAL; 			// logitude of Geo positions		"posLon":{"value":<POS_LON>}
	(* Process Value *)                 		                            		
	xMotorOn          		: BOOL;				// Status Motor On					"motorOn":{"value":<MOTOR_ON>},	
	xRightLeft          	: BOOL;				// Direction of the Motor			"rightLeft":{"value":<RIGHT_LEFT>},
	rCurrent            	: REAL; 			// Current in A						"current":{"value":<CURRENT>,"unit":"A"},
	rEnergy            		: REAL; 			// energy in kWh					"energy":{"value":<ENERGY>,"unit":"kWh"},
	rThermalMotorImage  	: REAL; 			// Tempeture in %,					"thermalMotorImage":{"value":<THERMAL_MOTOR_IMAGE>,"unit":"%%"},
	rTemperature       		: REAL; 			// Tempeture in °C,					"temperature":{"value":<TEMPERATURE>,"unit":"°C"},
	wErrorCode      		: WORD;				// Error Code 						"errorCode":{"value":<ERROR_CODE>},	
	dwSwitchCycles			: DWORD;			// Switch Cycles for right 			"switchCycles":{"value":<SWITCH_CYCLES>},
	dwSwitchCyclesLeft		: DWORD;			// Switch Cycles for Left 			"switchCyclesLeft":{"value":<SWITCH_CYCLES_LEFT>},
	dwRuntime				: DWORD; 			// Time in s						"runtime":{"value":<RUNTIME>,"unit":"s"},
	dwIdletime				: DWORD; 			// Time in s						"idletime":{"value":<IDLE_TIME>,"unit":"s"},
    dwTriptime 				: DWORD; 			// Time in s						"triptime":{"value":<TRIP_TIME>,"unit":"s"},
	(*Parameter Values from PKE und Drive*)
	byClass    				: BYTE;				// Class Value form PKE	 			"class":{"value":<CLASS>},  
    rOverloadReleaseIr 		: REAL; 			// adjust Overload Value PKE		"overloadReleaseIr":{"value":<OVERLAOD_RELEASE_IR>,"unit":"A"},
    rFreqMax  				: REAL; 			// Parameter Drive					"freqMax":{"value":<FREQ_MAX>,"unit":"Hz"},
    rFreqMin 				: REAL; 			// Parameter Drive					"freqMin":{"value":<FREQ_MIN>,"unit":"Hz"},
    rTimeAcc 				: REAL; 			// Parameter Drive					"timeAcc":{"value":<TIME_ACC>,"unit":"s"},
    rTimeDec 				: REAL; 			// Parameter Drive					"timeDec":{"value":<TIME_DEC>,"unit":"s"},
    rMotorNomVolt 			: REAL; 			// Parameter Drive					"motorNomVolt":{"value":<MOTOR_NOM_VOLT>,"unit":"V"},
    rMotorNomCurr 			: REAL; 			// Parameter Drive					"motorNomCurr":{"value":<MOTOR_NOM_CURR>,"unit":"A"},
    rMotorNomFreq 			: REAL; 			// Parameter Drive					"motorNomFreq":{"value":<MOTOR_NOM_FREQ>,"unit":"Hz"},
    rMotorNomSpeed 			: REAL; 			// Parameter Drive					"motorNomSpeed":{"value":<MOTOR_NOM_SPEED>,"unit":"rpm"}
	(*Device Managment Information from the CMS *)
	strMotorName			: STRING; 			// motor identifier in the app 		"motorName":{"value":0,"type":"STRING","string":"<MOTOR_NAME>"},
	(*Device Managment Information from the Part Protection*)
	eProtTypecode 			: teProtTypecode; 	// Typecode	(see enum) 				"protTypecode":{"value":<PROT_TYPE_CODE>},
	strProtSupplier			: STRING; 			// Supplier Name					"protSupplier":{"value":0,"type":"STRING","string":"<PROT_SUPPLIER"},
	strProtOrderNum			: STRING; 			// Order Number						"protOrderNumber":{"value":0,"type":"STRING","string":"<PROT_ORDER_NUMBER>"},
	strProtProductionDate	: STRING; 			// Producation Date					"protProductionDate":{"value":0,"type":"STRING","string":"<PROT_PRODUCTION_DATE>"}	
	(*Device Managment Information from the Part Starter*)
	eStartTypecode    		: teStartTypecode;	// Typecode	(see enum)				"startTypecode":{"value":<START_TYPECODE>},
	eStartConn				: teFieldbus;		// Fieldbus connection				"startConn":{"value":<START_CONN>},
	strStartSupplier		: STRING; 	  		// Supplier Name					"startSupplier":{"value":0,"type":"STRING","string":"<START_SUPPLIER>"},
	strStartOrderNum		: STRING; 			// Order Number						"startOrderNumber":{"value":0,"type":"STRING","string":"<START_ORDER_NUMBER>"},
	strStartProductionDate	: STRING; 			// Producation Date					"startProductionDate":{"value":<START_PRODUCTION_DATE>},
	strStartFirmwareVersion	: STRING; 			// Firmware Version 				"startFirmwareVersion":{"value":0,"type":"STRING","string":"<START_FIRMWARE_VERSION"},
	(*Device Managment Information from the Part "3rd party" 
	e.g. Motor, Incoder, Temperature Sensor *)
	str3rdTypeCode			: STRING; 			// text string specifiying device 	"3rdTypecode":{"value":0,"type":"STRING","string":"<3RD_TYPECODE>"},
	str3rdSupplier			: STRING;			// Supplier Name					"3rdSupplier":{"value":0,"type":"STRING","string":"<3RD_SUPPLIER>"},
	str3rdOrderNumber		: STRING; 			// OrderNumber from Supplier		"3rdOrderNumber":{"value":0,"type":"STRING","string":"<3RD_ORDER_NUMBER>"},
	str3rdProductionDate	: STRING;  			// Producation Date from Device		"3rdProductionDate":{"value":<3RD_PRODUCTION_DATE>},
	str3rdFirmwareVer		: STRING;			// Firmware Version from Device		"3rdFirmwareVersion":{"value":0,"type":"STRING","string":"<3RD_FIRMWARE_VERSION>"},
	str3rdSerialNum			: STRING; 			// Serial Number from Device		"3rdSerialNumber":{"value":0,"type":"STRING","string":"<3RD_SERIAL_NUMBER>"}
 
END_STRUCT
END_TYPE

// Structs/tsProtectionDevicInfo
(*Device Managment Information from the Part Protection*)
TYPE tsProtectionDevicInfo :
STRUCT		
	eProtTypecode 			: teProtTypecode; 	// Typecode	(see enum) 				
	strProtSupplier			: STRING; 			// Supplier Name					
	strProtOrderNum			: STRING[20]; 		// Order Number						
	strProtProductionDate	: STRING[20]; 		// Producation Date					
END_STRUCT
END_TYPE

// Structs/tsStarterDevicInfo
(*Device Managment Information from the Part Starter*)
TYPE tsStarterDevicInfo :
STRUCT		
	eStartTypecode    		: teStartTypecode;	// Typecode	(see enum)				
	eStartConn				: teFieldbus;		// Fieldbus connection				
	strStartSupplier		: STRING; 	  		// Supplier Name					
	strStartOrderNum		: STRING[20]; 		// Order Number						
	strStartProductionDate	: STRING[20]; 		// Producation Date					
	strStartFirmwareVersion	: STRING[20]; 		// Firmware Version 				
END_STRUCT                                                                          
END_TYPE

// Basic/Enums/teFieldbus
{attribute 'qualified_only'}
{attribute 'strict'}
//Fieldbus connectivty from Eaton Device for Motor Starter
TYPE teFieldbus :
(
	unknown 		:= 0, //unknown 
	ModbusRTU		:= 1, //ModbusRTU	
	ModbusTCP		:= 2, //ModbusTCP		
	SWD				:= 3, //SWD		
	Profibus		:= 4, //Profibus		
	Profinet		:= 5, //Profinet		
	DeviceNet		:= 6, //DeviceNet	
	EthernetIP		:= 7, //EthernetIP
	EtherCat		:= 8  //EtherCat
)WORD;
END_TYPE

// Basic/Enums/teProtTypecode
{attribute 'qualified_only'}
{attribute 'strict'}
//Typcode from Eaton Device for Motor Protection
TYPE teProtTypecode :
(
	Nothing := 0,	//Nothing 
	PKZ		:= 1,   //PKZ - Motor Protective Circuit Breakers mechanic	   
	PKE		:= 2,   //PKE - Motor Protective Circuit Breakers electronic		   
	NZM		:= 3    //NZM - Moulded Case Circuit Breaker		   
)WORD;
END_TYPE

// Basic/Enums/teStartTypecode
{attribute 'qualified_only'}
{attribute 'strict'}
//Typcode from Eaton Device for Motor Starter
TYPE teStartTypecode :
(
	Nothing := 0, // Nothing 
	DIL		:= 1, // DIL - contactor	
	EMS		:= 2, // EMS - electronic Motor Starter		
	DC1		:= 3, // DC1 - compact Drive		
	DE1		:= 4, // DE1 - variable Speed Starter		
	DA1		:= 5, // DA1 - advanced Drive		
	DG1		:= 6, // DG1 - general purpose Drive	
	DIUL	:= 7, // DIUL - reversing contactor
	DS7		:= 8  // DS7 - Softstarter
)WORD;
END_TYPE

// Structs/DA1/teDriveError
{attribute 'qualified_only'}
//Definition from Error Code which are come from Eaton Drives
TYPE teDriveError :
(	
 no_Flt  		:=0,  //Shown FOR P0-13 IF there are no messages in the error register.									DA1, DC1, DE1
 OI_b 			:=1,  //Excessively high braking current                                                                   DA1, DC1, DE1
 OL_br 			:=2,  //Thermal overload on brake resistor.                                                                DA1, DC1, DE1
 O_I 			:=3,  //Overcurrent AT variable frequency drive output                                                     DA1, DC1, DE1
 It_trP 		:=4,  //Motor overload.                                                                                    DA1, DC1, DE1
 PS_trp 		:=5,  //Overcurrent (Hardware)                                                                             DA1, DC1, DE1
 OVolt 			:=6,  //Overvoltage in DC link                                                                             DA1, DC1, DE1
 VVolt 			:=7,  //Undervoltage in DC link.                                                                           DA1, DC1, DE1
 O_t 			:=8,  //Overtemperature AT heat sink.                                                                      DA1, DC1, DE1
 V_t 			:=9,  //Under-temperature                                                                                  DA1, DC1, DE1
 P_dEf 			:=10,  //The parameters‘ default settings have been loaded.                                                 DA1, DC1, DE1
 E_trip 		:=11,  //External Fault                                                                                     DA1, DC1, DE1
 SC_ObS 		:=12,  //Communication error with an external operating unit OR with a PC                                   DA1, DC1, DE1
 FlT_dc 		:=13,  //Excessively high DC link voltage ripple                                                            DA1, DC1, DE1
 P_LOss 		:=14,  //Incoming power phase failure (only FOR devices with a three-phase power supply)                    DA1, DC1, DE1
 h_O_I 			:=15,  //Overcurrent AT output, DC1 motor pick-up control fault												DA1, DE1 
 Th_flt 		:=16,  //Malfunctioning heat sink thermistor.																DA1, DC1, DE1
 dAtA_F 		:=17,  //Error in INTERNAL memory                                                                           DA1, DC1, DE1
 F_4_20 		:=18,  	//The analog input's input current does not fall within the specified range.                        DA1, DC1, DE1
 dAtA_E 		:=19,  //Error in internal memory																			DA1, DC1…E1
 V_dEf 			:=20,  //The customer'S settings FOR the parameters have been imported.										DA1 
 F_Ptc 			:=21,  //Motor PTC thermistor overtemperature																DA1, DC1…E1 
 FAn_F 			:=22,  //The device‘S INTERNAL fan is experiencing a fault                                                  DA1, DC1…E1 
 O_hEAt 		:=23,  //The measured ambient temperature exceeds the specified value.                                      DA1, DC1…E1 
 O_torQ 		:=24,  //Maximum permissible torque exceeded.																DA1 		
 U_torQ 		:=25,  //Only active IF brake control is enabled in hoisting gear mode (P2-18 = 8).							DA1
 OUt_F   		:=26,  //Device output fault                                                                     			DA1, DC1…E1
 Sto_F 			:=29,  //Internal STO circuit fault                                                                    		DA1 
 Enc_01 		:=30,  //No communication between the encoder module and the variable frequency drive                  		DA1 
 Enc_02 		:=31,  //The calculated motor speed is different from the measured motor speed                         		DA1 
 Enc_03 		:=32,  //The motor speed and the PPR value entered in P6-06 do not match.                              		DA1 
 Enc_04 		:=33,  //Channel A fault                                                                               		DA1 
 Enc_05 		:=34,  //Channel B fault                                                                               		DA1 
 Enc_06 		:=35,  //Error on channels A and B                                                                     		DA1 
 AtF_01 		:=40,  //Motor identification failed																		DA1, DC1…E1 
 AtF_02 		:=41,  //Motor identification failed: The measured stator resistance is too large.                          DA1, DC1…E1 
 AtF_03 		:=42,  //Motor identification failed: The measured motor inductance is too low.                             DA1, DC1…E1 
 AtF_04 		:=43,  //Motor identification failed: The measured motor inductance is too high.                            DA1, DC1…E1 
 AtF_05 		:=44,  //Motor identification failed: The measured motor parameters do not match.                           DA1, DC1…E1 
 Out_Ph 		:=49,  //A phase in the motor cable is not connected or has a discontinuity.                                DA1, DC1…E1 
 Sc_FO1 		:=50,  //No valid Modbus frame was received within the time specified.                                      DA1, DC1…E1 
 Sc_FO2 		:=51,  //No valid CANopen frame was received within the specified time.                                     DA1, DC1…E1 
 Sc_FO3 		:=52,  //Communications between the device and the plugged-in field bus option have dropped out.			DA1 
 Sc_F04 		:=53,  //Communications between the device and the plugged-in I/O expansion have dropped out.          		DA1 
 OF_01 			:=60,  //No internal connection to an optional card                                                    		DA1 
 OF_02 			:=61,  //Optional module in abnormal state                                                             		DA1 
 PLC_01 		:=70,  //Non-supported function block from function block editor                                       		DA1 
 PLC_02 		:=71,  //Program from function block editor is too big                                                 		DA1 
 PLC_03 		:=72,  //Division by zero                                                                              		DA1 
 PLC_04 		:=73,  //Lower limit is higher than upper limit                                                        		DA1 
 PLC_05 		:=74   //Overflow table Function block editor                                                          		DA1 *)
)BYTE;
END_TYPE

// Structs/DA1/teDriveParameter
{attribute 'qualified_only'}
{attribute 'strict'}
//Definition of available Parameter from drive
TYPE teDriveParameter :
(
AnalogInput1		,// 20 P0-01 Analog Input 1 ro – 4096 ≙ 100.0 % U16
AnalogInput2		,// 21 P0-02 Analog Input 2 ro – 4096 ≙ 100.0 % U16
DIstatus 			,// 11 P0-03 DI status ro – Bit 0 ≙ digital input 1 Bit 1 ≙ digital input 2 … WORD
fPreRamp 			,// 22 P0-04 f-PreRamp ro – S16
TorqueRef 			,// 41 P0-05 Torque Reference ro – 1000 ≙ 100.0 % U16
MotorPotRef			,// 42 P0-06 MotorPot Reference ro – U16 
MotorTorque 		,//  9 P0-12 Motor Torque ro – 1000 ≙ 100.0 % U16
DCLinkVoltage 		,// 23 P0-20 DC-Link Voltage ro – 600 ≙ 600 V
HeatsinkTemp 		,// 24 P0-21 Heatsink Temperature ro – 40 ≙ 40 °C
kWhMeter			,// 30 P0-26 kWh Meter ro – 100 ≙ 10.0 kWh U16
MWhMeter  			,// 33 P0-27 MWh Meter ro – U16
tRun				,// 34 P0-31 t-Run ro – U16
tMinSec				,// 35 P0-31 t-min/sec ro – U16
tHoursRun			,// 36 P0-34 t-HoursRun Enable ro – U16	
fmax				,//101 P1-01 f-max rw RUN 3000 ≙ 50.0 Hz P1-02 - (5 x P1-09)(max.: 500.0 Hz /30000 rpm)U16
fmin				,//102 P1-02 f-min rw RUN 3000 ≙ 50.0 Hz 0.0 Hz - P1-01 U16
tacc				,//103 P1-03 t-acc rw RUN 300 ≙ 30.0 s 0.00 s - 6000 s U16
tdec				,//104 P1-04 t-dec rw RUN 300 ≙ 30.0 s 0.00 s - 6000 s U16
StopMode			,//105 P1-05 Stop Mode rw RUN – 0, 1, 2, 3, 4 U16
EnergyOptimizer		,//106 P1-06 EnergyOptimizer rw RUN – 0, 1 WORD
MotorNomVoltage 	,//107 P1-07 Motor Nom Voltage rw STOP 230 ≙ 230 V 0 - Ue U16
MotorNomCurrent 	,//108 P1-08 Motor Nom Current rw STOP 1 ≙ 0.1 A (0.1 - 1) x Ie U16
MotorNomFreq 		,//109 P1-09 Motor Nom Frequency rw STOP 50 ≙ 50 Hz 10 Hz - 500 Hz U16
MotorNomSpeed 		,//110 P1-10 Motor Nom Speed rw RUN 1500 ≙ 1500 rpm • 0• 200 - 30000 rpm U16
VBoost				,//111 P1-11 V-Boost rw STOP -1 ≙ Auto0 ≙ Disabled 1 ≙ 0.1 % • 0: Auto • 0 - 30.0 % of P1-07 S16
LocalProcessData	,//112 P1-12 Local ProcessData Source rw STOP – 0 - 13 U16
DIConfig			,//113 P1-13 DI Config Select rw STOP – 0 - 21 U16
fFix1				,//201 P2-01 f-Fix1 rw RUN 3000 ≙ 50.0 Hz P1-02 (min: 0 Hz / 0 rpm) - P1-01 (max: 500.0 Hz / 30000 rpm) U16
fFix2				,//202 P2-02 f-Fix2 rw RUN 3000 ≙ 50.0 Hz P1-02 (min: 0 Hz / 0 rpm) - P1-01 (max: 500.0 Hz / 30000 rpm) U16
fFix3				,//203 P2-03 f-Fix3 rw RUN 3000 ≙ 50.0 Hz P1-02 (min: 0 Hz / 0 rpm) - P1-01 (max: 500.0 Hz / 30000 rpm) U16
fFix4				,//204 P2-04 f-Fix4 rw RUN 3000 ≙ 50.0 Hz P1-02 (min: 0 Hz / 0 rpm) - P1-01 (max: 500.0 Hz / 30000 rpm) U16
fFix5				,//205 P2-05 f-Fix5 rw RUN 3000 ≙ 50.0 Hz P1-02 (min: 0 Hz / 0 rpm) - P1-01 (max: 500.0 Hz / 30000 rpm) U16
fFix6				,//206 P2-06 f-Fix6 rw RUN 3000 ≙ 50.0 Hz P1-02 (min: 0 Hz / 0 rpm) - P1-01 (max: 500.0 Hz / 30000 rpm) U16
fFix7				,//207 P2-07 f-Fix7 rw RUN 3000 ≙ 50.0 Hz P1-02 (min: 0 Hz / 0 rpm) - P1-01 (max: 500.0 Hz / 30000 rpm) U16
fFix8				 //208 P2-08 f-Fix8 rw RUN 3000 ≙ 50.0 Hz P1-02 (min: 0 Hz / 0 rpm) - P1-01 (max: 500.0 Hz / 30000 rpm) U16
);
END_TYPE

// Structs/DA1/teDriveTyp
{attribute 'qualified_only'}
//Definition of possible Eaton Drive Types
TYPE teDriveTyp :(
	DE1 	:=8, 		//variable speed starter
	DC1 	:=10, 		//compact drive
	DA1		:=5632, 	//advanced drive
	DE11 	:=9			//new version from De1 variable speed starter
	)WORD;
END_TYPE

// Structs/DA1/tsCommandAndControl16bit
//Control Word Structure from Drive, with this Comands the Drive can be controlled
{attribute 'analysis' := '-33, -12'} 
{attribute 'naming' := 'off'} 
TYPE tsCommandAndControl16bit :
STRUCT	
	Operation		: BIT; //False = stop; 								TRUE = Operation
	Direction		: BIT; //False = Clockwise rotating field (FWD); 	TRUE = Anticlockwise rotating field (REV)
	ResetFault		: BIT; //False = No action,							TRUE = Fault Reset
	FreeRunDown		: BIT; //False = No action,							TRUE = free run-down
	bit5			: BIT; //Not used        							
	QuickStop		: BIT; //False = No action,							TRUE = Quick stop (ramp)
	FixedFrequencq	: BIT; //False = No action,							TRUE = Fixed frequency 1 (FF1)
	SetpointToZero	: BIT; //False = No action,							TRUE = Overwrite setpoint value with 0
	bit9			: BIT; //Not used
	bit10			: BIT; //Not used
	bit11			: BIT; //Not used
	bit12			: BIT; //Not used
	bit13			: BIT; //Not used
	bit14			: BIT; //Not used
	bit15			: BIT; //Not used
	bit16			: BIT; //Not used
	
END_STRUCT
END_TYPE

// Structs/DA1/tsDriveCommandAndSpeed
//Union for Hardware Mapping from Register to Comand and Control Structure
TYPE tsDriveCommandAndSpeed :
STRUCT	
	stCommandDrive	: tsCommandAndControl16bit;	//Command Structure from Drive
	iSpeedReference	: INT;							//Speed Reference  from Drive
END_STRUCT	
END_TYPE

// Structs/DA1/tsDriveStatusAndSpeed
//Union for Hardware Mapping from Register to Status Structure
TYPE tsDriveStatusAndSpeed :
STRUCT
	stStatusDrive	: tsStatusAndFaults16bit;	//Status Structure from Drive
	iMotorSpeed		: INT;						//Motor Speed from Drive
	iCurrent		: INT;						//Current from Drive
END_STRUCT
END_TYPE

// Structs/DA1/tsStatusAndFaults16bit
//Status Structure from Drive
{attribute 'analysis' := '-12'} 
{attribute 'naming' := 'off'} 
TYPE tsStatusAndFaults16bit :
STRUCT
		
	Readiness		: BIT;				//False = Drive not ready; 						TRUE = ready FOR operation (READY)
	Operation		: BIT;              //False = stop; 								TRUE = Operation (RUN)
	Rotation		: BIT;              //False = Clockwise rotating field (FWD),		TRUE = Anticlockwise rotating field (REV)
	Fault			: BIT;              //False = no error,								TRUE = Fault detected (FAULT)
	SetpointReached	: BIT;              //False = Acceleration ramp 					TRUE = Frequency actual value equals setpoint input       							
	ZeroSpeed		: BIT;              //False = -,									TRUE = Zero speed
	SpeedControl	: BIT;              //False = Speed control deactivated,			TRUE = Speed control activated
	HardwareEnable	: BIT;              //False = No coomunication,						TRUE = communication and Hardware okay
	ErrorCode		: teDriveError;		//Detailed Error Information Code

END_STRUCT
END_TYPE

// Structs/SWD/tePkeProfile
{attribute 'qualified_only'}
{attribute 'strict'}
//Different Profile which are available in PKE with SWD
TYPE tePkeProfile :
(
	eProfile1 := 1,	//Profile 1 has 2 Input Bytes
	eProfile2 := 2,	//Profile 2 has 4 Input Bytes
	eProfile3 := 3	//Profile 3 has 5 Input Bytes
);
END_TYPE

// Structs/SWD/tsIB0_PKE_SWD_32
//First Status Byte from PKE Swd in Profil 3
{attribute 'conditionalshow'}
TYPE tsIB0_PKE_SWD_32 :
STRUCT
	bit0ContactorState 				: BIT;		// Status of Contactor	
    bit1PkeStatus 					: BIT;		// Status of Pke
    bit2SwitchManualOnOff			: BIT;		//Position of 1-0-A switch 	00: Incorrect position for longer than 4 seconds
	bit3SwitchPosManualAuto			: BIT;		//							01: Position A (Switching command via SWD)
												//							10: Position 0 (Contactor OFF)
												//							11: Position 1 (Contactor ON)
    bit4GroupDiagnostic 			: BIT;		//0: No diagnostic alarm; 
    bit5Reserved 					: BIT;      // Reserved
    bit6ModulPresent 				: BIT;      //0: module not present; 1: module present
    bit7SUBST						: BIT;      //0: configured module present; 1: universal module M22-SWD-NOP(C) present
END_STRUCT
END_TYPE

// Structs/SWD/tsIB1_PKE_SWD_32
//Extended Status Information from PKE Byte 1 
{attribute 'conditionalshow'}
TYPE tsIB1_PKE_SWD_32 :
STRUCT
	bit0SetValueIr0 			: BIT;		//Set value Ir
    bit1SetValueIr1 			: BIT;		//Set value Ir
    bit2SetValueIr2 	  		: BIT;		//Set value Ir
    bit3SetValueIr3 			: BIT;		//Set value Ir
    bit4TripReason0 			: BIT;		//Trip reason
    bit5TripReason1 			: BIT;		//Trip reason
    bit6TripReason2 			: BIT;		//Trip reason
    bit7AckZmrRequired			: BIT;		//ZMR manual function acknowledgement required
											//0: No acknowledgement required; 1: Acknowledgement of overload required
END_STRUCT
END_TYPE

// Structs/SWD/tsIB4_PKE_SWD_32
//Idendifikation Byte 4 from SWD PKE Profil 3
{attribute 'conditionalshow'}
TYPE tsIB4_PKE_SWD_32 :
STRUCT
	bit0PartTripBlock0 			: BIT;	//3 bits used for coding Trip Block 
    bit1PartTripBlock1 			: BIT;	//3 bits used for coding Trip Block
    bit2PartTripBlock2 	  		: BIT;	//3 bits used for coding Trip Block
    bit3SetTimeLag0 			: BIT;	//3 bits used for coding the Psotion from Time Lag Switch
    bit4SetTimeLag1 			: BIT;	//3 bits used for coding the Psotion from Time Lag Switch
    bit5SetTimeLag2 			: BIT;	//3 bits used for coding the Psotion from Time Lag Switch
    bit6Reserved 				: BIT;	//Reserved
    bit7Reserved				: BIT;	//Reserved
END_STRUCT
END_TYPE

// Structs/SWD/tsIB_DIL_SWD_32
//Definition of contactor DIL SWD Modul
{attribute 'conditionalshow'}
TYPE tsIB_DIL_SWD_32 :
STRUCT
	bit0ContactorState 		: BIT;			// Status of Contactor	
    bit1X1_X2 				: BIT;			//0: Auxiliary contact for X1-X2 opened 1: Auxiliary contact for X1-X2 closed
											//The meaning depends on the auxiliary contact used.
    bit2X1_X0 	  			: BIT;			//0: Auxiliary contact for X1-X0 opened 1: Auxiliary contact for X1-X0 closed
											//The meaning depends on the auxiliary contact used.
    bit3SwitchManualOnOff	: BIT; 			//0: Automatic; 1: Manual mode State can be read in first bit
    bit4GroupDiagnostic 	: BIT;			//0: No diagnostic alarm; 
    bit5Reserved6 			: BIT;			// Reserved
    bit6ModulPresent 		: BIT;			//0: module not present; 1: module present
    bit7SUBST				: BIT;			//0: configured module present; 1: universal module M22-SWD-NOP(C) present
END_STRUCT
END_TYPE

// Structs/SWD/tsPKE_ModXTUA
//Structure from PKE Profil 3
{attribute 'conditionalshow'}
TYPE tsPKE_ModXTUA :
STRUCT
	wTripUnit 			: WORD; //(TYPE) [encoded] (see 27)	FROM 0 TO 9
	wSetValueIr 		: WORD; //[encoded] (see 26)	from 0 to 15
	wCLASS 				: WORD; //– Set time lag [encoded] (see 0)	from 0 to 4
	wPkeStatus 			: WORD; //PKE ON/OFF	0 or 1
	wTripReason 		: WORD; //[encoded] (see 42)	from 0 to 4 
	wThermalMotorImage 	: WORD; //[%] (see 36)	from 0 (0%) to 120 (120%)
	wSetValueIrA 		: WORD; //[human readable format]	1.2 unit, 330mA = 33, 1200mA = 120 ( divided by 100/scaling factor 100)
	wCLASS_s 			: WORD; //– Set time lag [human readable value]	5, 10, 15, 20, 99-test trip / CP 50, 65, 80 (divided by 10) 99-test trip  
	wCurrent			: WORD; //Relative current value of the highest phase current [%] only XTUA  	120 (120%)
	wCurrentA			: WORD; //Relative current value of the highest phase current [human readable format] only XTUA  	1.2 unit, 330mA = 33 ( divided by 100)
END_STRUCT
END_TYPE

// Structs/SWD/tsPKE_Profil1
//Structure from PKE Profil 3
{attribute 'conditionalshow'}
TYPE tsPKE_Profil1 :
STRUCT
	stInputBy0 	: tsIB0_PKE_SWD_32;	//Status Information
	stInputBy1 	: tsIB1_PKE_SWD_32;	//Status Information
END_STRUCT
END_TYPE

// Structs/SWD/tsPKE_Profil2
//Structure from PKE Profil 3
{attribute 'conditionalshow'}
TYPE tsPKE_Profil2 :
STRUCT
	stInputBy0 	: tsIB0_PKE_SWD_32;	//Status Information
	stInputBy1 	: tsIB1_PKE_SWD_32;	//Status Information
	byInputBy2 	: BYTE; 			//Motor current [%]
	byInputBy3 	: BYTE; 			//Thermal motor image [%]
END_STRUCT
END_TYPE

// Structs/SWD/tsPKE_Profil3
//Structure from PKE Profil 3
{attribute 'conditionalshow'}
TYPE tsPKE_Profil3 :
STRUCT
	stInputBy0 	: tsIB0_PKE_SWD_32;	//Status Information
	stInputBy1 	: tsIB1_PKE_SWD_32;	//Status Information
	byInputBy2 	: BYTE; 			//Motor current [%]
	byInputBy3 	: BYTE; 			//Thermal motor image [%]
	stInputBy4 	: tsIB4_PKE_SWD_32;	//Identification 
END_STRUCT
END_TYPE

// Structs/SWD/tsQB_DIL_SWD_32
// Output Structure from DIL SWD modul
{attribute 'conditionalshow'}
TYPE tsQB_DIL_SWD_32 :
STRUCT
	bit0Contactor 		: BIT;		//Contactor Switch On or OFF
    bit1Reserved 		: BIT;      //Reserved 
    bit2Reserved 		: BIT;      //Reserved 
    bit3Reserved 		: BIT;      //Reserved 
    bit4Reserved 		: BIT;      //Reserved 
    bit5Reserved 		: BIT;      //Reserved 
    bit6Reserved 		: BIT;      //Reserved 
    bit7Reserved		: BIT;      //Reserved 
END_STRUCT
END_TYPE

// Structs/SWD/tsQB_PKE_Mod
//Output Structure from PKE on SWD
{attribute 'conditionalshow'}
TYPE tsQB_PKE_Mod :
STRUCT
	byResetAvg		: BYTE; // Reset AVG/MAX values in data flash
	byResetCounter	: BYTE; // Reset all trip counters
	byRemoteTrip	: BYTE; //R-TRIP Remote tripping, PKE basic device 0: no remote tripping 1: Remote tripping
END_STRUCT
END_TYPE

// Structs/SWD/tsQB_PKE_SWD_32
//Output Structure from PKE on SWD
{attribute 'conditionalshow'}
TYPE tsQB_PKE_SWD_32 :
STRUCT
	bit0Contactor 		: BIT;		//Contactor Switch On or OFF
    bit0Reserved 		: BIT;		//Reserved
    bit2ZmrOnOff 		: BIT;		//activate ZMR Function
    bit3ZMRAutoHand		: BIT;		//Mode of ZMR; in auto Mode Motor will start automatically in manual 
    bit4Reserved 		: BIT;		//Reserved
    bit5Reserved 		: BIT;		//Reserved
    bit6Reserved 		: BIT;		//Reserved
    bit7Reserved		: BIT;		//Reserved
END_STRUCT
END_TYPE

// Basic/Enums/Error/teErrorCodeEaton
// Error Code Definition
{attribute 'analysis' := '-13'}
TYPE teErrorCodeEaton :
(
	//General Configuration Error
	NoError 			:= 0, 	//No Error
	WrongConfig			:= 1,	//Wrong or missing configuration of Inputs
	FieldbusComError	:= 7, 	//Fieldbus Communication Error to the Motor Devices
	MasterComErr		:= 8,  	//Fieldbus Master Communication Error	
	InpAddressMiss		:= 9,  	//Input  Address from Device is missing
	OutAddressMiss		:= 10,  //Output Address from Device is missing
	DeviceMissing		:= 11,  //Device Address is missing	
	WrongDevice			:= 12,  //Wrong Device connect; isn't a PKE		
	ComErrIntern		:= 13,	//No communication between PKESWD-32 AND PKE trip block
	
	
	//Drive Error with offset 100
	OI_b 				:=101,  //Excessively high braking current                                                                   DA1, DC1, DE1
	OL_br 				:=102,  //Thermal overload on brake resistor.                                                                DA1, DC1, DE1
	O_I 				:=103,  //Overcurrent AT variable frequency drive output                                                     DA1, DC1, DE1
	It_trP 				:=104,  //Motor overload.                                                                                    DA1, DC1, DE1
	PS_trp 				:=105,  //Overcurrent (Hardware)                                                                             DA1, DC1, DE1
	OVolt 				:=106,  //Overvoltage in DC link                                                                             DA1, DC1, DE1
	VVolt 				:=107,  //Undervoltage in DC link.                                                                           DA1, DC1, DE1
	O_t 				:=108,  //Overtemperature AT heat sink.                                                                      DA1, DC1, DE1
	V_t 				:=109,  //Under-temperature                                                                                  DA1, DC1, DE1
	P_dEf 				:=110,  //The parameters‘ default settings have been loaded.                                                 DA1, DC1, DE1
	E_trip 				:=111,  //External Fault                                                                                     DA1, DC1, DE1
	SC_ObS 				:=112,  //Communication error with an external operating unit OR with a PC                                   DA1, DC1, DE1
	FlT_dc 				:=113,  //Excessively high DC link voltage ripple                                                            DA1, DC1, DE1
	P_LOss 				:=114,  //Incoming power phase failure (only for devices with a three-phase power supply)                    DA1, DC1, DE1
	h_O_I 				:=115,  //Overcurrent at output, DC1 motor pick-up control fault												DA1, DE1 
	Th_flt 				:=116,  //Malfunctioning heat sink thermistor.																DA1, DC1, DE1
	dAtA_F 				:=117,  //Error in internal memory                                                                           DA1, DC1, DE1
	F_4_20 				:=118,  //The analog input's input current does not fall within the specified range.                        DA1, DC1, DE1
	dAtA_E 				:=119,  //Error in internal memory																			DA1, DC1…E1
	V_dEf 				:=120,  //The customer's settings for the parameters have been imported.										DA1 
	F_Ptc 				:=121,  //Motor PTC thermistor overtemperature																DA1, DC1…E1 
	FAn_F 				:=122,  //The device‘S INTERNAL fan is experiencing a fault                                                  DA1, DC1…E1 
	O_hEAt 				:=123,  //The measured ambient temperature exceeds the specified value.                                      DA1, DC1…E1 
	O_torQ 				:=124,  //Maximum permissible torque exceeded.																DA1 		
	U_torQ 				:=125,  //Only active if brake control is enabled in hoisting gear mode (P2-18 = 8).							DA1
	OUt_F   			:=126,  //Device output fault                                                                     			DA1, DC1…E1
	Sto_F 				:=129,  //Internal STO circuit fault                                                                    		DA1 
	Enc_01 				:=130,  //No communication between the encoder module and the variable frequency drive                  		DA1 
	Enc_02 				:=131,  //The calculated motor speed is different from the measured motor speed                         		DA1 
	Enc_03 				:=132,  //The motor speed and the PPR value entered in P6-06 do not match.                              		DA1 
	Enc_04 				:=133,  //Channel A fault                                                                               		DA1 
	Enc_05 				:=134,  //Channel B fault                                                                               		DA1 
	Enc_06 				:=135,  //Error on channels A and B                                                                     		DA1 
	AtF_01 				:=140,  //Motor identification failed																		DA1, DC1…E1 
	AtF_02 				:=141,  //Motor identification failed: The measured stator resistance is too large.                          DA1, DC1…E1 
	AtF_03 				:=142,  //Motor identification failed: The measured motor inductance is too low.                             DA1, DC1…E1 
	AtF_04 				:=143,  //Motor identification failed: The measured motor inductance is too high.                            DA1, DC1…E1 
	AtF_05 				:=144,  //Motor identification failed: The measured motor parameters do not match.                           DA1, DC1…E1 
	Out_Ph 				:=149,  //A phase in the motor cable is not connected or has a discontinuity.                                DA1, DC1…E1 
	Sc_FO1 				:=150,  //No valid Modbus frame was received within the time specified.                                      DA1, DC1…E1 
	Sc_FO2 				:=151,  //No valid CANopen frame was received within the specified time.                                     DA1, DC1…E1 
	Sc_FO3 				:=152,  //Communications between the device and the plugged-in field bus option have dropped out.			DA1 
	Sc_F04 				:=153,  //Communications between the device and the plugged-in I/O expansion have dropped out.          		DA1 
	OF_01 				:=160,  //No internal connection to an optional card                                                    		DA1 
	OF_02 				:=161,  //Optional module in abnormal state                                                             		DA1 
	PLC_01 				:=170,  //Non-supported function block from function block editor                                       		DA1 
	PLC_02 				:=171,  //Program from function block editor is too big                                                 		DA1 
	PLC_03 				:=172,  //Division by zero                                                                              		DA1 
	PLC_04 				:=173,  //Lower limit is higher than upper limit                                                        		DA1 
	PLC_05 				:=174,   //Overflow table Function block editor                                                          		DA1 *)	

	//General SWD Error
	SwitchErr			:=200,	//No unambiguous position OF the 1-0-A switch FOR more than 4 seconds
	
	//Special PKE Error with offset 300
	Overload 			:=201, 	//PKE has switched off
	ShortCircuit		:=202, 	//PKE has switched off
	PhaseFailure		:=203, 	//Disconnection at: 100 % of the thermal motor image (TH)
	TestPosition		:=204, 	//Test position on PKEXTU(W)A-…
	OverloadWithZMR		:=205, 	//Überlastfall mit aktivierter ZMR-Funktion Leistungsschütz hat abgeschaltet, der Wert des thermischen Motorabbildes (TH) ist nach der Abschaltung noch größer als 100 %
	RemoteTripping		:=206, 	//Remote tripping through output bit
	SwitchOff			:=207,	//PKZ tripped position or PKE is switchoff from hand
	ContactorStick		:=208	//Contactor sticks
	
) INT;
END_TYPE

// Basic/Enums/PKE/teCurrentUnit
//Different Unit Option in PKE to read current Value
{attribute 'qualified_only'}
{attribute 'strict'}
TYPE teCurrentUnit :
(
	Percent ,		// current in % - based on the set max current value
	Ampere ,		// Unit for Current is A
	mAmpere 		// Unit for Current is mA
);
END_TYPE

// Basic/Enums/PKE/tePkeErrorCode
//Trip Reason from PKE 
//hide symbol of teTripReason are neccessary because teTripReason is internal enum from Hardware and will be displayed in this summary enum for End user
{attribute 'analysis' := '-13'}
TYPE tePkeErrorCode :
(
	NotDefined 			:= 0, 	//No Error
	Overload 			:= 1, 	//PKE has switched off
	ShortCircuit		:= 2, 	//PKE has switched off
	PhaseFailure		:= 3, 	//Disconnection at: 100 % of the thermal motor image (TH)
	TestPosition		:= 4, 	//Test position on PKEXTU(W)A-…
	OverloadWithZMR		:= 5, 	//Überlastfall mit aktivierter ZMR-Funktion Leistungsschütz hat abgeschaltet, der Wert des thermischen Motorabbildes (TH) ist nach der Abschaltung noch größer als 100 %
	RemoteTripping		:= 6, 	//Remote tripping through output bit
	FieldbusComError	:= 7, 	//Fieldbus Communication Error to the Motor Devices
	ManualTripping		:= 8,	//Manual Tripping form switch in PKE
	MasterComErr		:= 9,  	//Fielbus Master Communication Error	
	InpAdressMiss		:= 10,  //Input Address from Device is missing
	OutAdressMiss		:= 11,  //Output Address from Device is missing
	DeviceMissing		:= 12,  //Device Address is missing	
	WrongDevice			:= 13,  // Wrong Device connect; isn't a PKE		
	ComErrIntern		:= 14,	//No communication between PKESWD-32 AND PKE trip block
	SwitchErr			:= 15	//No unambiguous position OF the 1-0-A switch FOR more than 4 seconds
)USINT;
END_TYPE

// Basic/Enums/PKE/teSwitchPos_1_0_A
//Position of Contactor Switch on SWD Modul
TYPE teSwitchPos_1_0_A :
(
	WrongPositiionLonger4sec 	:= 0,	//Not allowed Postion longer 4 sec
	PosA_CommandSWD 			:= 1,	// Position is on A this allowed the control of contactor over SWD from PLC
	Pos0_ContactorOFF			:= 2,	// Contactor every time off Output from SWD will be ignore
	Pos1_ContactorON			:= 3	// Contactor every time on Output from SWD will be ignore
)USINT;
END_TYPE

// Basic/Enums/PKE/teTripBlock
//Definition of the different Types of Trip BLock from PKE
TYPE teTripBlock :
(
	PKE_XTUA_1_2 	:= 0,	//Max Current 1.2 A
	PKE_XTUA_4		:= 1,	//Max Current 4 A
	PKE_XTUA_12 	:= 2,	//Max Current 12 A
	PKE_XTUA_32		:= 3	//Max Current 32 A
)WORD;
END_TYPE

// Basic/Enums/PKE/teTripReason
//Trip Reason from PKE 
TYPE teTripReason :
(
	NotDefined 			:= 0, //Status not defined
	Overload 			:= 1, //PKE has switched off
	ShortCircuit		:= 2, //PKE has switched off
	PhaseFailure		:= 3, //Disconnection at: 100 % of the thermal motor image (TH)
	TestPosition		:= 4, //Test position on PKEXTU(W)A-…
	OverloadWithZMR		:= 5, //Überlastfall mit aktivierter ZMR-Funktion Leistungsschütz hat abgeschaltet, der Wert des thermischen Motorabbildes (TH) ist nach der Abschaltung noch größer als 100 %
	RemoteTripping		:= 6,  //Remote tripping through output bit
	ManualTripping		:= 7	//Manual switch from Maintenace guy
)USINT;
END_TYPE

// Global Variables/GVL_Const
VAR_GLOBAL CONSTANT
	MAX_Observer : UINT := 20;
END_VAR

VAR_GLOBAL
	aritfObserver : ARRAY [0..GVL_Const.MAX_Observer]OF IBasicBehaviour;
END_VAR

// Global Variables/GVL_ErrorCodeDefEaton
{attribute 'qualified_only'}
VAR_GLOBAL CONSTANT
	//General Configuration Error
	NoError 			:INT :=  0; 	//No ErrorEND_VAR
	WrongConfi			:INT :=  1;	//Wrong or missing configuration of Inputs
	FieldbusComError	:INT :=  7; 	//Fieldbus Communication Error to the Motor Devices
	MasterComErr		:INT :=  8;  	//Fielbus Master Communication Error	
	InpAdressMiss		:INT :=  9;  	//Input Address from Device is missing
	OutAdressMiss		:INT := 10;  //Output Address from Device is missing
	DeviceMissing		:INT := 11;  //Device Address is missing	
	WrongDevice			:INT := 12;  //Wrong Device connect; isn't a PKE		
	ComErrIntern		:INT := 13;	//No communication between PKESWD-32 AND PKE trip block

	
	//Drive Error with offset 100
	OI_b 				: INT :=101;  //Excessively high braking current                                                                   DA1, DC1, DE1
	OL_br 				: INT :=102;  //Thermal overload on brake resistor.                                                                DA1, DC1, DE1
	O_I 				: INT :=103;  //Overcurrent AT variable frequency drive output                                                     DA1, DC1, DE1
	It_trP 				: INT :=104;  //Motor overload.                                                                                    DA1, DC1, DE1
	PS_trp 				: INT :=105;  //Overcurrent (Hardware)                                                                             DA1, DC1, DE1
	OVolt 				: INT :=106;  //Overvoltage in DC link                                                                             DA1, DC1, DE1
	VVolt 				: INT :=107;  //Undervoltage in DC link.                                                                           DA1, DC1, DE1
	O_t 				: INT :=108;  //Overtemperature AT heat sink.                                                                      DA1, DC1, DE1
	V_t 				: INT :=109;  //Under-temperature                                                                                  DA1, DC1, DE1
	P_dEf 				: INT :=110;  //The parameters‘ default settings have been loaded.                                                 DA1, DC1, DE1
	E_trip 				: INT :=111;  //External Fault                                                                                     DA1, DC1, DE1
	SC_ObS 				: INT :=112;  //Communication error with an external operating unit OR with a PC                                   DA1, DC1, DE1
	FlT_dc 				: INT :=113;  //Excessively high DC link voltage ripple                                                            DA1, DC1, DE1
	P_LOss 				: INT :=114;  //Incoming power phase failure (only FOR devices with a three-phase power supply)                    DA1, DC1, DE1
	h_O_I 				: INT :=115;  //Overcurrent AT output, DC1 motor pick-up control fault												DA1, DE1 
	Th_flt 				: INT :=116;  //Malfunctioning heat sink thermistor.																DA1, DC1, DE1
	dAtA_F 				: INT :=117;  //Error in INTERNAL memory                                                                           DA1, DC1, DE1
	F_4_20 				: INT :=118;  //The analog input's input current does not fall within the specified range.                        DA1, DC1, DE1
	dAtA_E 				: INT :=119;  //Error in internal memory																			DA1, DC1…E1
	V_dEf 				: INT :=120;  //The customer'S settings FOR the parameters have been imported.										DA1 
	F_Ptc 				: INT :=121;  //Motor PTC thermistor overtemperature																DA1, DC1…E1 
	FAn_F 				: INT :=122;  //The device‘S INTERNAL fan is experiencing a fault                                                  DA1, DC1…E1 
	O_hEAt 				: INT :=123;  //The measured ambient temperature exceeds the specified value.                                      DA1, DC1…E1 
	O_torQ 				: INT :=124;  //Maximum permissible torque exceeded.																DA1 		
	U_torQ 				: INT :=125;  //Only active IF brake control is enabled in hoisting gear mode (P2-18 = 8).							DA1
	OUt_F   			: INT :=126;  //Device output fault                                                                     			DA1, DC1…E1
	Sto_F 				: INT :=129;  //Internal STO circuit fault                                                                    		DA1 
	Enc_01 				: INT :=130;  //No communication between the encoder module and the variable frequency drive                  		DA1 
	Enc_02 				: INT :=131;  //The calculated motor speed is different from the measured motor speed                         		DA1 
	Enc_03 				: INT :=132;  //The motor speed and the PPR value entered in P6-06 do not match.                              		DA1 
	Enc_04 				: INT :=133;  //Channel A fault                                                                               		DA1 
	Enc_05 				: INT :=134;  //Channel B fault                                                                               		DA1 
	Enc_06 				: INT :=135;  //Error on channels A and B                                                                     		DA1 
	AtF_01 				: INT :=140;  //Motor identification failed																		DA1, DC1…E1 
	AtF_02 				: INT :=141;  //Motor identification failed: The measured stator resistance is too large.                          DA1, DC1…E1 
	AtF_03 				: INT :=142;  //Motor identification failed: The measured motor inductance is too low.                             DA1, DC1…E1 
	AtF_04 				: INT :=143;  //Motor identification failed: The measured motor inductance is too high.                            DA1, DC1…E1 
	AtF_05 				: INT :=144;  //Motor identification failed: The measured motor parameters do not match.                           DA1, DC1…E1 
	Out_Ph 				: INT :=149;  //A phase in the motor cable is not connected or has a discontinuity.                                DA1, DC1…E1 
	Sc_FO1 				: INT :=150;  //No valid Modbus frame was received within the time specified.                                      DA1, DC1…E1 
	Sc_FO2 				: INT :=151;  //No valid CANopen frame was received within the specified time.                                     DA1, DC1…E1 
	Sc_FO3 				: INT :=152;  //Communications between the device and the plugged-in field bus option have dropped out.			DA1 
	Sc_F04 				: INT :=153;  //Communications between the device and the plugged-in I/O expansion have dropped out.          		DA1 
	OF_01 				: INT :=160;  //No internal connection to an optional card                                                    		DA1 
	OF_02 				: INT :=161;  //Optional module in abnormal state                                                             		DA1 
	PLC_01 				: INT :=170;  //Non-supported function block from function block editor                                       		DA1 
	PLC_02 				: INT :=171;  //Program from function block editor is too big                                                 		DA1 
	PLC_03 				: INT :=172;  //Division by zero                                                                              		DA1 
	PLC_04 				: INT :=173;  //Lower limit is higher than upper limit                                                        		DA1 
	PLC_05 				: INT :=174;  //Overflow table Function block editor                                                          		DA1 *)	

	//General SWD Error
	SwitchErr			: INT :=200;	//No unambiguous position OF the 1-0-A switch FOR more than 4 seconds
	
	//Special PKE Error with offset 300
	Overload 			: INT :=201; 	//PKE has switched off
	ShortCircuit		: INT :=202; 	//PKE has switched off
	PhaseFailure		: INT :=203; 	//Disconnection at: 100 % of the thermal motor image (TH)
	TestPosition		: INT :=204; 	//Test position on PKEXTU(W)A-…
	OverloadWithZMR		: INT :=205; 	//Überlastfall mit aktivierter ZMR-Funktion Leistungsschütz hat abgeschaltet, der Wert des thermischen Motorabbildes (TH) ist nach der Abschaltung noch größer als 100 %
	RemoteTripping		: INT :=206; 	//Remote tripping through output bit
END_VAR

// Device/Application/PLC_PRG
PROGRAM PLC_PRG
VAR

	
	MyMotor : FB_Drive;
	MyMotor2 : FB_Drive;
	xEnable : BOOL := TRUE;
	xOn: BOOL;
	rVelocity: REAL;
	xSwitchDC1: BOOL := TRUE;
	itfDrive : ITF_Drive := MyMotor2;
	ErrorHandler : FB_ErrorHandler;
	xTest : Bool;
END_VAR

IF xSwitchDC1 THEN
	itfDrive := MyMotor;	
ELSE
	itfDrive := MyMotor2;
END_IF

itfDrive.Operation := xOn;
itfDrive.rVelocity := rVelocity;

	MyMotor(
		xDone=> , 
		xBusy=> , 
		xError=> , 
		xEnable:= xEnable, 
		itfHW_Node:= Modbus_Slave_DC1, 
		eErrorCode=> );

	MyMotor2(
		xDone=> , 
		xBusy=> , 
		xError=> , 
		xEnable:= xEnable, 
		itfHW_Node:= Modbus_Slave_DA1, 
		eErrorCode=> );


ErrorHandler(astrActive=> , uiNumOfActError=> );

END_PROGRAM

// XV300/Application/PLC_PRG
PROGRAM PLC_PRG
VAR	
	MyPke		: FB_PKE;
	ePkeError	: teErrorCodeEaton;
	rCurrentPKE	: REAL;
	xEnable		: BOOL := TRUE;
	xOn			: BOOL;
END_VAR


MyPke(
	xDone=> , 
	xBusy=> , 
	xError=> , 
	xEnable:= xEnable, 
	itfHW_Node:= MainMotor, 
	eErrorCode=> ePkeError);

rCurrentPKE := MyPke.Current_A;
MyPke.Contactor := xOn;

END_PROGRAM

// FunctionBlock/FB_PKE
//FB which handle the Communicatution with a Hardware PKE from Eaton
//{attribute 'conditionalshow_all_locals'}
FUNCTION_BLOCK FB_PKE EXTENDS FB_HWDeviceBasic IMPLEMENTS ITF_DIL, ITF_PKE
VAR
	//Access to HW IO
	_pstPkeProfil3	: POINTER TO tsPKE_Profil3;			//Input Byte from PKE Profil 3
	_pstPkeProfil2	: POINTER TO tsPKE_Profil2;			//Input Byte from PKE Profil 2
	_pstPkeProfil1	: POINTER TO tsPKE_Profil1;			//Input Byte from PKE Profil 1
	_pstPkeOutput 	: POINTER TO tsQB_PKE_SWD_32;		//Output Byte from PKE Profil 1-3	
	_pstModInp 		: POINTER TO tsPKE_ModXTUA;			//Input Structure from Modbus XTUA first 10 Register
	_pstModOut 		: POINTER TO tsQB_PKE_Mod;			//Output Coil from PKE Modubs RTU	
	
	//Loal Status Information from PKE
	_ePkeProfile					: tePkeProfile; //read actual Profile from Device Description Parameter 2200000102
	_xContactorState 				: BOOL;				// Status of Contactor	
    _xPKE_Status 					: BOOL;				// Status of Pke
	_eConSwitchState 				: teSwitchPos_1_0_A;//Contactor manual Switch Psoition
	_rSelectValueIr 				: REAL;				//Set value Ir
	_eTripReason 					: teTripReason;		//Trip reason
	_xAckZMR_manualRequired			: BOOL; 			//ZMR manual function acknowledgement required
	_byMotorCurrent 				: BYTE; 			//Motor current [%]
	_byMotorImage 					: BYTE; 			//Thermal motor image [%]
	
    _bySetTimeLag 					: BYTE;				//3 bits used for coding the Psotion from Time Lag Switch
	_xContactor						: BOOL;				//Switch Contactor On or OFF
	_xOverloadProtectionZMR 		: BOOL;				//Settings for ZMR Function
	_xZMR_AutoHand 					: BOOL;				//Mode of ZMR; in auto Mode Motor will start automatically in manual
	_xResetAvg						: BOOL;				// Reset Avg Values
	_xRemoteTrip					: BOOL;				// Remote Trip
	_xResetCounter					: BOOL;				// Reset Trip Counters on Asic 
	_ePartTipBlock					: teTripBlock;		// Used Trip Block in PKE HW
	//Device Information Parameter
	_strDeviceCode					: STRING(51);	// Hardware Version Name from Device read acyclic
    _xSUBST							: BOOL;      	//0: configured module present; 1: universal module M22-SWD-NOP(C) present	
    _xGroupDiagnostic 				: BOOL;			//0: No diagnostic alarm; 
    _xModulPresent 					: BOOL;      	//0: module not present; 1: module present	
	//{if defined (XV303)}
	_ModuleInfo 		: EA_SWD.GetModuleInfo;								// FB for SWD for read some Module Info
	_ModuleDiagInfo 	: EA_SWD.struct_SWD_MODULEDIAG;						// structure for Diagnostic Value	
	//{end_if}	
END_VAR
VAR_STAT CONSTANT
	//Table to now the Max Current Value from Version and Switch Position
	c_arCurrentIr : ARRAY[0..15, 0..3] OF REAL := 		[0.30, 1.00,  3.00,  8.00,
                                                      	0.33, 1.10,  3.30,  8.80,
                                                        0.36, 1.20,  3.60,  9.70,
   							                            0.40, 1.30,  4.00, 10.50,
   							                            0.43, 1.42,  4.30, 11.50,
   							                            0.47, 1.55,  4.70, 12.50,
   							                            0.50, 1.70,  5.00, 13.50,
   							                            0.56, 1.90,  5.60, 15.00,
   							                            0.63, 2.10,  6.30, 17.00,
   							                            0.70, 2.40,  7.00, 19.00,
   							                            0.77, 2.60,  7.70, 20.50,
   							                            0.83, 2.80,  8.30, 22.00,
   							                            0.90, 3.00,  9.00, 24.00,
   							                            1.00, 3.30, 10.00, 27.00,
   							                            1.10, 3.70, 11.00, 29.00,
   							                            1.20, 4.00, 12.00, 32.00];


END_VAR

SUPER^();

{attribute 'monitoring' := 'variable'}
//Acknowledge required for ZMR Function
PROPERTY ACKR : BOOL
GET
// Implemntation of get 
{attribute 'analysis' := '-162'}
ACKR := _xAckZMR_manualRequired;
END_GET
SET
_xZMR_AutoHand := ACKR;
END_SET
END_PROPERTY

ACTION ACT_MapModbus:
//Map SWD Pke value from Hardware structure to local Variable
(*IF _pstModInp <> 0 THEN		
	{attribute 'analysis' := '-34, -130'} //this Action is for mapping values from fieldbus to end user udt
	_xPKE_Status 		:= _pstModInp^.wPkeStatus.0;
	IF _pModbusRTUSlave <> 0 THEN
		_xModulPresent 		:= _pModbusRTUSlave^.xInitDone;	
	END_IF							
	_ePartTipBlock 		:= _pstModInp^.wTripUnit; 		
	_rSelectValueIr 	:= c_arCurrentIr[_ePartTipBlock ,_pstModInp^.wSetValueIr ];				
	_eTripReason 		:= WORD_TO_BYTE(_pstModInp^.wTripReason);				
	_byMotorCurrent 	:= WORD_TO_BYTE(_pstModInp^.wCurrent);			
	_byMotorImage 		:= WORD_TO_BYTE(_pstModInp^.wThermalMotorImage);						
	_bySetTimeLag 		:= WORD_TO_BYTE(_pstModInp^.wCLASS); 
END_IF	
IF _pstModOut <> 0 THEN		
	_pstModOut^.byResetAvg		:= BOOL_TO_BYTE(_xResetAvg);	
	_pstModOut^.byResetCounter 	:= BOOL_TO_BYTE(_xResetCounter);
	_pstModOut^.byRemoteTrip 	:= BOOL_TO_BYTE(_xRemoteTrip);		
END_IF*)
END_ACTION

ACTION ACT_MapSWD:
//Map SWD Pke value from Hardware structure to local Variable
IF _pstPkeProfil3 <> 0 THEN
	{attribute 'analysis' := '-34, -130'} //this Action is for mapping values from fieldbus to end user udt
	_xContactorState  	:= _pstPkeProfil3^.stInputBy0.bit0ContactorState;			
	_xPKE_Status 		:= _pstPkeProfil3^.stInputBy0.bit1PkeStatus;	
	_xModulPresent 		:= _pstPkeProfil3^.stInputBy0.bit6ModulPresent;								
	_xGroupDiagnostic 	:= _pstPkeProfil3^.stInputBy0.bit4GroupDiagnostic;	
	_xSUBST				:= _pstPkeProfil3^.stInputBy0.bit7SUBST;	
	_eConSwitchState 	:= ( SHL (BIT_TO_BYTE (_pstPkeProfil3^.stInputBy0.bit3SwitchPosManualAuto), 1)) OR (BIT_TO_BYTE (_pstPkeProfil3^.stInputBy0.bit2SwitchManualOnOff));	
	_rSelectValueIr 	:= c_arCurrentIr[ (( SHL (BIT_TO_BYTE (_pstPkeProfil3^.stInputBy1.bit3SetValueIr3), 3)) OR ( SHL (BIT_TO_BYTE (_pstPkeProfil3^.stInputBy1.bit2SetValueIr2), 2)) OR ( SHL (BIT_TO_BYTE (_pstPkeProfil3^.stInputBy1.bit1SetValueIr1), 1)) OR (BIT_TO_BYTE (_pstPkeProfil3^.stInputBy1.bit0SetValueIr0))),_ePartTipBlock ];				
	_eTripReason 		:= ( SHL (BIT_TO_BYTE (_pstPkeProfil3^.stInputBy1.bit6TripReason2), 2)) OR ( SHL (BIT_TO_BYTE (_pstPkeProfil3^.stInputBy1.bit5TripReason1), 1)) OR (BIT_TO_BYTE (_pstPkeProfil3^.stInputBy1.bit4TripReason0));			
	_xAckZMR_manualRequired	:= _pstPkeProfil3^.stInputBy1.bit7AckZmrRequired;		
	_byMotorCurrent 	:= _pstPkeProfil3^.byInputBy2;			
	_byMotorImage 		:= _pstPkeProfil3^.byInputBy3;	
	_ePartTipBlock 		:= ( SHL (BIT_TO_BYTE (_pstPkeProfil3^.stInputBy4.bit2PartTripBlock2), 2)) OR ( SHL (BIT_TO_BYTE (_pstPkeProfil3^.stInputBy4.bit1PartTripBlock1), 1)) OR (BIT_TO_BYTE (_pstPkeProfil3^.stInputBy4.bit0PartTripBlock0)); 							
	_bySetTimeLag 		:= ( SHL (BIT_TO_BYTE (_pstPkeProfil3^.stInputBy4.bit5SetTimeLag2), 2)) OR ( SHL (BIT_TO_BYTE (_pstPkeProfil3^.stInputBy4.bit4SetTimeLag1), 1)) OR (BIT_TO_BYTE (_pstPkeProfil3^.stInputBy4.bit3SetTimeLag0)); 
ELSIF _pstPkeProfil2 <> 0 THEN
	{attribute 'analysis' := '-34, -130'} //this Action is for mapping values from fieldbus to end user udt
	_xContactorState  	:= _pstPkeProfil2^.stInputBy0.bit0ContactorState;			
	_xPKE_Status 		:= _pstPkeProfil2^.stInputBy0.bit1PkeStatus;	
	_xModulPresent 		:= _pstPkeProfil2^.stInputBy0.bit6ModulPresent;								
	_xGroupDiagnostic 	:= _pstPkeProfil2^.stInputBy0.bit4GroupDiagnostic;	
	_xSUBST				:= _pstPkeProfil2^.stInputBy0.bit7SUBST;	
	_eConSwitchState 	:= ( SHL (BIT_TO_BYTE (_pstPkeProfil2^.stInputBy0.bit3SwitchPosManualAuto), 1)) OR (BIT_TO_BYTE (_pstPkeProfil2^.stInputBy0.bit2SwitchManualOnOff));	
	_rSelectValueIr 	:= c_arCurrentIr[ (( SHL (BIT_TO_BYTE (_pstPkeProfil2^.stInputBy1.bit3SetValueIr3), 3)) OR ( SHL (BIT_TO_BYTE (_pstPkeProfil2^.stInputBy1.bit2SetValueIr2), 2)) OR ( SHL (BIT_TO_BYTE (_pstPkeProfil2^.stInputBy1.bit1SetValueIr1), 1)) OR (BIT_TO_BYTE (_pstPkeProfil2^.stInputBy1.bit0SetValueIr0))),_ePartTipBlock ];				
	_eTripReason 		:= ( SHL (BIT_TO_BYTE (_pstPkeProfil2^.stInputBy1.bit6TripReason2), 2)) OR ( SHL (BIT_TO_BYTE (_pstPkeProfil2^.stInputBy1.bit5TripReason1), 1)) OR (BIT_TO_BYTE (_pstPkeProfil2^.stInputBy1.bit4TripReason0));			
	_xAckZMR_manualRequired	:= _pstPkeProfil2^.stInputBy1.bit7AckZmrRequired;		
	_byMotorCurrent 	:= _pstPkeProfil2^.byInputBy2;			
	_byMotorImage 		:= _pstPkeProfil2^.byInputBy3;	
ELSIF _pstPkeProfil1 <> 0 THEN
	{attribute 'analysis' := '-34, -130'} //this Action is for mapping values from fieldbus to end user udt
	_xContactorState  	:= _pstPkeProfil1^.stInputBy0.bit0ContactorState;			
	_xPKE_Status 		:= _pstPkeProfil1^.stInputBy0.bit1PkeStatus;	
	_xModulPresent 		:= _pstPkeProfil1^.stInputBy0.bit6ModulPresent;								
	_xGroupDiagnostic 	:= _pstPkeProfil1^.stInputBy0.bit4GroupDiagnostic;	
	_xSUBST				:= _pstPkeProfil1^.stInputBy0.bit7SUBST;	
	_eConSwitchState 	:= ( SHL (BIT_TO_BYTE (_pstPkeProfil1^.stInputBy0.bit3SwitchPosManualAuto), 1)) OR (BIT_TO_BYTE (_pstPkeProfil1^.stInputBy0.bit2SwitchManualOnOff));	
	_rSelectValueIr 	:= c_arCurrentIr[ (( SHL (BIT_TO_BYTE (_pstPkeProfil1^.stInputBy1.bit3SetValueIr3), 3)) OR ( SHL (BIT_TO_BYTE (_pstPkeProfil1^.stInputBy1.bit2SetValueIr2), 2)) OR ( SHL (BIT_TO_BYTE (_pstPkeProfil1^.stInputBy1.bit1SetValueIr1), 1)) OR (BIT_TO_BYTE (_pstPkeProfil1^.stInputBy1.bit0SetValueIr0))),_ePartTipBlock ];				
	_eTripReason 		:= ( SHL (BIT_TO_BYTE (_pstPkeProfil1^.stInputBy1.bit6TripReason2), 2)) OR ( SHL (BIT_TO_BYTE (_pstPkeProfil1^.stInputBy1.bit5TripReason1), 1)) OR (BIT_TO_BYTE (_pstPkeProfil1^.stInputBy1.bit4TripReason0));			
	_xAckZMR_manualRequired	:= _pstPkeProfil1^.stInputBy1.bit7AckZmrRequired;		
END_IF	
IF _eTripReason = teTripReason.NotDefined AND NOT _xPKE_Status THEN
	_eTripReason := teTripReason.ManualTripping;
END_IF
IF _pstPkeOutput <> 0 THEN		
	_pstPkeOutput^.bit0Contactor	:= _xContactor;	
	_pstPkeOutput^.bit2ZmrOnOff := _xOverloadProtectionZMR;
	_pstPkeOutput^.bit3ZMRAutoHand := _xZMR_AutoHand;		
END_IF
END_ACTION

//Class Information from PKE, time delay
PROPERTY Class : BYTE
GET
// Implemntation of get 
{attribute 'analysis' := '-162'}
Class := _bySetTimeLag;
END_GET
END_PROPERTY

//Status and Control Contactor
PROPERTY Contactor : BOOL
GET
// Implemntation of get 
{attribute 'analysis' := '-162'}
Contactor := _xContactorState;
END_GET
SET
_xContactor := Contactor;
END_SET
END_PROPERTY

//Current in A 
{attribute 'monitoring' := 'variable'}
PROPERTY Current_A : REAL
GET
// Implemntation of get 
{attribute 'analysis' := '-162'}
Current_A := BYTE_TO_REAL(_byMotorCurrent)/100.0 * SelectValueIr;
END_GET
END_PROPERTY

//Mapped real Hardware IO from GVL_IO to definied internal Structure and Interface
{attribute 'naming' := 'omit'} 
METHOD CyclicAction
VAR_INPUT
	{attribute 'analysis' := '-33'} 
	itfTimingController	: CBML.ITimingController; //Timing Controller for Check Time Out
END_VAR
VAR_OUTPUT
	//if xComplete or iErrorID <> 0 then the CleanupAction is reached
	xComplete	: BOOL;								//Normally never use
	iErrorID	: INT;								//Error is happen, Error Code 
END_VAR
//Call Cyclic Action form Device Base for standard error handling
SUPER^.CyclicAction(itfTimingController := itfTimingController ,xComplete=>xComplete, iErrorID =>iErrorID);

//Device specific error code
IF _eTripReason <> teTripReason.NotDefined THEN	
	{analysis -34, -58} //map device specific error code to a eaton uniqe global error code: offset for pke is 200
	IF _eTripReason = teTripReason.ManualTripping THEN
		eErrorCode := teErrorCodeEaton.RemoteTripping;
	ELSE
		eErrorCode := TO_INT(_eTripReason + 200);	
	END_IF
	{analysis +34, +58}	
END_IF

//Special Handling for different Fieldbus System
CASE _eBusType OF
	DED.BUS_TYPE.MODBUS_RTU:
			ACT_MapModbus();
	DED.BUS_TYPE.VEN_SPEC:
			ACT_MapSWD();
			{IF defined (variable: _ModuleInfo)}
			_ModuleInfo(
					xExecute:= , 
					byModuleNo:= _byModulAddress,  
					sProductName=> _strDeviceCode, 
				);
			IF _xGroupDiagnostic THEN
				IF EA_SWD.GetModuleDiag (byModuleNo := _byModulAddress, pSwdModuleDiag := ADR(_ModuleDiagInfo)) THEN
					IF _ModuleDiagInfo.xExtendedDiagAvailable THEN
						CASE _ModuleDiagInfo.abyExtendedDiag[1] OF
							16#03 : eErrorCode := teErrorCodeEaton.ComErrIntern;
							16#15 : eErrorCode := teErrorCodeEaton.SwitchErr;
						END_CASE
					END_IF	
				END_IF		
			ELSE
				_ModuleDiagInfo.xExtendedDiagAvailable := FALSE;
			END_IF
			{END_IF}
END_CASE
END_METHOD

//Detail Error Code from PKE
PROPERTY ErrorCode : teErrorCodeEaton
GET
// Implemntation of get 
{attribute 'analysis' := '-162'}
ErrorCode := eErrorCode;
END_GET
END_PROPERTY

//Give the Current back in the defined Unit 
METHOD M_Current : REAL
VAR_INPUT
	eCurrentUnit : teCurrentUnit;	//Define the Unit of the Return Value
END_VAR
CASE eCurrentUnit OF
	teCurrentUnit.Percent: 
			IF _pstPkeProfil3 <> 0 THEN
				M_Current := BYTE_TO_REAL(_pstPkeProfil3^.byInputBy2);
			ELSE
				M_Current := 0;	
			END_IF	
	teCurrentUnit.Ampere: M_Current := Current_A;
	teCurrentUnit.mAmpere: M_Current := Current_A *1000;
	ELSE  M_Current := 0.0;
END_CASE
END_METHOD

//Identification Modul Name
{attribute 'analysis' := '-23'} 
PROPERTY ModulName : STRING[51]
GET
// Implemntation of get 
{attribute 'analysis' := '-23-, 162'}
ModulName := _strDeviceCode;
END_GET
END_PROPERTY

//Modul Present on SWD
PROPERTY ModulPresent : BOOL
GET
// Implemntation of get 
{attribute 'analysis' := '-162'}
ModulPresent := _xModulPresent;
END_GET
END_PROPERTY

// Information of Connection Status on Fieldbus
PROPERTY P_xConnected  : BOOL
GET
// Implemntation of get 
{attribute 'analysis' := '-162'}
P_xConnected := (_DeviceState = DED.DEVICE_STATE.RUNNING);
END_GET
END_PROPERTY

//Error happen on Device
PROPERTY P_xError : BOOL
GET
// Implemntation of get 
{attribute 'analysis' := '-162'}
P_xError := _xGroupDiagnostic OR NOT _xPKE_Status OR (_DeviceState = DED.DEVICE_STATE.ERROR) OR xError;
END_GET
END_PROPERTY

{attribute 'monitoring' := 'variable'}
//Install Trip Block
PROPERTY PartTripBlock : teTripBlock
GET
// Implemntation of get 
{attribute 'analysis' := '-162'}
PartTripBlock  := _ePartTipBlock;
END_GET
END_PROPERTY

//Status from PKE
PROPERTY PkeStatus : BOOL
GET
PkeStatus := _xPKE_Status;
END_GET
END_PROPERTY

//Defined Max Ir Value
PROPERTY SelectValueIr : REAL
GET
// Implemntation of get 
{attribute 'analysis' := '-162'}
SelectValueIr := _rSelectValueIr;
END_GET
END_PROPERTY

//Initalization Routine
(*Init for Drive FB*)
{attribute 'naming' := 'omit'} 
METHOD StartAction
VAR_OUTPUT
	xComplete	: BOOL;		//Setting and Init Done, if the Variable is True the Method Cyclic will be called
	iErrorID	: INT;		//if Error is happen set ErrorID to Error Code, after that CLeanUp will Call with Error ID as an Input
END_VAR
VAR
	_pConfigParam 	: POINTER TO IoConfigParameter;	//Pointer to a Parameter from DeviceDescription
	_pPointerValue	: POINTER TO BYTE;				//Pointer to a Value in the Device Description
	_udiResult 		: UDINT;						//Result from Function to read Parameters					
END_VAR
//Call Start Action form Device Base
SUPER^.StartAction(xComplete=>xComplete, iErrorID =>iErrorID);

//Check if In and Output is set
//Read the Parameter for the IO input pointer which is generate in the special devicedescription
_pConfigParam := IoStandard.ConfigGetParameter(pIoConnector:= _itfDevice.Connector, dwParameterId := 2147483649);
IF _pConfigParam <> 0 THEN
	_pbyInputAdress := IoStandard.ConfigGetParameterValuePointer(_pConfigParam, pResult:=ADR(_udiResult));
END_IF
_pConfigParam := IoStandard.ConfigGetParameter(pIoConnector:= _itfDevice.Connector, dwParameterId := 2200000102); //parameter for identifiy the Profile
IF _pConfigParam <> 0 THEN
	_pPointerValue := IoStandard.ConfigGetParameterValuePointer(_pConfigParam, pResult:=ADR(_udiResult));
	IF _pPointerValue <> 0 THEN
		IF _pPointerValue^ = 16#94 THEN
			_ePkeProfile := tePkeProfile.eProfile3;
		ELSIF _pPointerValue^ = 16#93 THEN
			_ePkeProfile := tePkeProfile.eProfile2;
		ELSIF _pPointerValue^ = 16#91 THEN
			_ePkeProfile := tePkeProfile.eProfile1;	
		END_IF
	END_IF
END_IF
IF _pbyInputAdress <> 0 THEN
	{analysis -19} //convert from input and output pointer to expected IO structure for PKE
	IF _eBusType = DED.BUS_TYPE.VEN_SPEC THEN
		IF    _ePkeProfile = tePkeProfile.eProfile3 THEN //Profile3
			_pstPkeProfil3 := _pbyInputAdress;
		ELSIF  _ePkeProfile = tePkeProfile.eProfile2 THEN //Profile2
			_pstPkeProfil2 := _pbyInputAdress;
		ELSIF  _ePkeProfile = tePkeProfile.eProfile1 THEN //Profile1
			_pstPkeProfil1 := _pbyInputAdress;	
		END_IF	
		{IF defined (variable: _ModuleInfo)}					
		_ModuleInfo.xExecute := TRUE;
		{END_IF}
	ELSIF _eBusType = DED.BUS_TYPE.MODBUS_RTU THEN
		_pstModInp := _pbyInputAdress;
	END_IF
ELSE
	eErrorCode := teErrorCodeEaton.InpAddressMiss; //wrong configuration
	iErrorID := TO_INT(eErrorCode);
END_IF

//Read the Parameter for the IO output pointer which is generate in the special devicedescription
_pConfigParam := IoStandard.ConfigGetParameter(pIoConnector:= _itfDevice.Connector, dwParameterId := 2147483648);
IF _pConfigParam <> 0 THEN
	_pbyOutputAdress := IoStandard.ConfigGetParameterValuePointer(_pConfigParam, pResult:=ADR(_udiResult));
END_IF
IF _pbyOutputAdress <> 0 THEN
	IF _eBusType = DED.BUS_TYPE.VEN_SPEC THEN
		_pstPkeOutput := _pbyOutputAdress;
	ELSIF _eBusType = DED.BUS_TYPE.MODBUS_RTU THEN
		_pstModOut := _pbyOutputAdress;
	END_IF	
	{analysis +19}		
ELSE
	eErrorCode := teErrorCodeEaton.OutAddressMiss; //wrong configuration 
	iErrorID := TO_INT(eErrorCode);
END_IF	
	
xComplete := TRUE;
END_METHOD

//Contactor manual Switch Psoition
{attribute 'monitoring' := 'variable'}
PROPERTY SwitchState_1_0_A : teSwitchPos_1_0_A
GET
// Implemntation of get 
{attribute 'analysis' := '-162'}
SwitchState_1_0_A  := _eConSwitchState;
END_GET
END_PROPERTY

//Thermal Motor Image calculate by Motor Protection
{attribute 'monitoring' := 'variable'}
PROPERTY ThermalMotorImage : REAL
GET
// Implemntation of get 
{attribute 'analysis' := '-162'}
ThermalMotorImage := BYTE_TO_REAL (_byMotorImage);
END_GET
END_PROPERTY

//Trip Reason 
{attribute 'monitoring' := 'variable'}
PROPERTY TripReason : teTripReason
GET
// Implemntation of get 
{attribute 'analysis' := '-162'}
TripReason := _eTripReason ;
END_GET
END_PROPERTY

//Set ZMR Mode to Auto or Hand
PROPERTY ZmrAutoHand : BOOL
GET
// Implemntation of get 
{attribute 'analysis' := '-162'}
ZmrAutoHand := _xZMR_AutoHand;
END_GET
SET
_xZMR_AutoHand := ZmrAutoHand;
END_SET
END_PROPERTY

END_FUNCTION_BLOCK

// Basic/FB/FB_HWDeviceBasic
//{attribute 'hide'}
//Basic FB for a HW Device 
{attribute 'reflection'}
FUNCTION_BLOCK FB_HWDeviceBasic EXTENDS FB_BasicWithBehaviour IMPLEMENTS I_HWDevice
VAR_INPUT
	xEnable 		: BOOL;			//	Activate the FB
	itfHW_Node 		: DED.INode;	
END_VAR
VAR_OUTPUT                                  	
	eErrorCode: teErrorCodeEaton;
END_VAR
VAR
	//Behaviour can be define here as a Dependicy Injection for Parent Groput
	_StateBehaviour 	: CBML.LConC;			//Define the Behaviour as LConC
	
	//Dependicy definet over FB_Init from user

  	_pbyInputAdress 		: POINTER TO BYTE;
 	_pbyOutputAdress 		: POINTER TO BYTE;
	
	//Device State and Information based on CAA Device Diagnostic Library
	_eBusType 			: DED.BUS_TYPE;		// Bus Type on which the Hardware is used
	_itfDevice 			: DED.IDevice;		// Interface to Device Information
	_itfParentDevice	: DED.IDevice;		// Interface to the Parent Device which is normally the Fieldbus Master
	_itfBus				: DED.IBus;			// Interface to Bus Information if this Fieldbus is upporting this Functonality
	_stDeviceInfo		: DED.DEVICE_INFO;	// stored Device Information which can be read with the Interface
	_stParentInfo		: DED.DEVICE_INFO;	// stored Fieldbus Master Device Information which can be read with the Interface
	_stBusInfo			: BUS_INFO;			// store Bus Information if it's available
	_DeviceState		: DEVICE_STATE;		// Device State in Device Tree
	_FieldbusMasterState: DEVICE_STATE;		// Parent Device State (Fieldbus Master)in Device Tree
	//Special Fielbus Information for differen Fieldbus Systems	
	_byModulAddress 	: BYTE;				//Hardware Adress from the Device in the Bussystem
	_wType				: WORD;				//Connector Type for identicate the Device if other information are not available	

	
	// The ID from Device Description to identify the Device
	_dwID: DWORD;
END_VAR

THIS^.IBehaviourModel := _StateBehaviour;
_StateBehaviour(xEnable:= xEnable, xBusy=> xBusy, xError=> xError);

//Mapped real Hardware IO from GVL_IO to definied internal Structure and Interface
{attribute 'naming' := 'omit'} 
METHOD CyclicAction
VAR_INPUT
	{attribute 'analysis' := '-33'} 
	itfTimingController	: CBML.ITimingController; //Timing Controller for Check Time Out
END_VAR
VAR_OUTPUT
	//if xComplete or iErrorID <> 0 then the CleanupAction is reached
	xComplete	: BOOL;								//Normally never use
	iErrorID	: INT;								//Error is happen, Error Code 
END_VAR
//Special Handling for different Fieldbus System
eErrorCode := teErrorCodeEaton.NoError;
CASE _eBusType OF
	DED.BUS_TYPE.MODBUS_RTU:
			;
	DED.BUS_TYPE.VEN_SPEC:
			;
END_CASE

//Check Device Status  from Tree; Device and Master
IF _itfDevice <> 0 THEN
	_DeviceState :=  _itfDevice.GetDeviceState();
END_IF
IF	_itfParentDevice <> 0 THEN
	_FieldbusMasterState := _itfParentDevice.GetDeviceState();
END_IF

IF _DeviceState <> DED.DEVICE_STATE.RUNNING THEN
	eErrorCode := teErrorCodeEaton.FieldbusComError;
END_IF

IF _FieldbusMasterState <> DED.DEVICE_STATE.RUNNING THEN
	eErrorCode := teErrorCodeEaton.MasterComErr;
END_IF
END_METHOD

//Information which kind of Fieldbus is in use
PROPERTY eFieldbus : teFieldbus
GET
CASE _eBusType OF
	//DED.BUS_TYPE.CANOPEN : eFieldbus := teFieldbus.CanOpen;
	DED.BUS_TYPE.MODBUS_RTU : eFieldbus := teFieldbus.ModbusRTU;
	DED.BUS_TYPE.MODBUS_TCP : eFieldbus := teFieldbus.ModbusTCP;
	DED.BUS_TYPE.VEN_SPEC : eFieldbus := teFieldbus.SWD;
	DED.BUS_TYPE.ETHERCAT : eFieldbus := teFieldbus.EtherCat;
END_CASE
END_GET
END_PROPERTY

//clean all values so that a restart is working fine again
METHOD ExitAction
VAR_INPUT
    xAfterCleanup : BOOL;
    xInCopyCode : BOOL;
END_VAR
	//Device State and Information based on CAA Device Diagnostic Library
	_eBusType 			:= DED.BUS_TYPE.UNKNOWN;		// Bus Type on which the Hardware is used
	_itfDevice 			:=0;		// Interface to Device Information
	_itfParentDevice	:=0;		// Interface to the Parent Device which is normally the Fieldbus Master
	_itfBus				:=0;			// Interface to Bus Information if this Fieldbus is upporting this Functonality
	//Special Fielbus Information for differen Fieldbus Systems	
	_byModulAddress 	:= 0;				//Hardware Adress from the Device in the Bussystem
	_DeviceState := DED.DEVICE_STATE.UNKNOWN;		
	_FieldbusMasterState	:= DED.DEVICE_STATE.UNKNOWN;
	_stBusInfo.eType := DED.BUS_TYPE.UNKNOWN;
	_stBusInfo.idInstance := 0;
	_stBusInfo.idSystem := 0;
END_METHOD

//Initalization Routine called from Runtime before Start
{attribute 'naming' := 'omit'} 
METHOD FB_Init : BOOL
VAR_INPUT
  bInitRetains : BOOL; // TRUE: the retain variables are initialized (reset warm / reset cold)
  bInCopyCode : BOOL;  // TRUE the instance will be copied to the copy-code afterward (online change)
END_VAR
VAR
	iIndex: INT;
END_VAR
FOR iIndex := 0 TO GVL_Const.MAX_Observer DO
	IF GVL_Const.aritfObserver[iIndex] = 0 THEN
		GVL_Const.aritfObserver[iIndex] := THIS^;
		EXIT;
	END_IF	
END_FOR
END_METHOD

//Initalization Routine
(*Init for Drive FB*)
{attribute 'naming' := 'omit'} 
METHOD StartAction
VAR_OUTPUT
	xComplete	: BOOL;		//Setting and Init Done, if the Variable is True the Method Cyclic will be called
	iErrorID	: INT;		//if Error is happen set ErrorID to Error Code, after that CLeanUp will Call with Error ID as an Input
END_VAR

VAR
	_itfFirstNode	 		: DED.INode;		//Interface from Hardware Device Tree
	_itfNextNode 			: DED.INode;		//Interface from Hardware Device Tree
	_itfParentNode 			: DED.INode;		//Interface from Hardware Device Tree
	_xRoot					: BOOL;				//Reached PLC as Root Level
	_udiSiblingNodeCount	: UDINT;			//Sibling Node Count in this Level; needed for found Modul Adress in SWD
	_udiLoop				: UDINT := 0;		//Help Varialble for Loops 
	_pConnector				: POINTER TO DED.IoConfigConnector; //Read Connector for information about Connector Type

END_VAR
{analysis -61, -46} // Querypointer used
//Check Bus System in which Device is running if _itfNode is set
IF itfHW_Node <> 0 THEN
	_itfParentNode := itfHW_Node.ParentNode;
	WHILE NOT _xRoot DO
		IF _itfParentNode <> 0 THEN
			_itfBus := DED.INode_TO_IBus(itfNode:= _itfParentNode);
			IF _itfBus <> 0 THEN
				//Get Bus Information
				_itfBus.GetBusInfo (buiInfo := _stBusInfo);
				_eBusType := _stBusInfo.eType;
				_itfParentDevice := DED.INode_TO_IDevice (itfNode := _itfParentNode);	//convert Prent Nod to Parent Device for diagnostic
				IF _itfParentDevice <> 0 THEN
					//read standard master infomation
					_itfParentDevice.GetDeviceInfo (deiInfo := _stParentInfo);
				END_IF
				_itfDevice:= DED.INode_TO_IDevice (itfNode := itfHW_Node);					//convert Node to Device for diagnostic
				IF _itfDevice <> 0 THEN
					//read standard device infomation
					_itfDevice.GetDeviceInfo (deiInfo := _stDeviceInfo);
					_pConnector := _itfDevice.Connector;
					_wType := _pConnector^.wType;	
				END_IF	
				EXIT;
			ELSIF _itfParentNode.IsRootNode THEN
				//No itfBus found in the Parent Node above the Input Node
				_xRoot := TRUE;
				_itfParentNode := itfHW_Node.ParentNode;	//set Parent Node over INode
				_itfParentDevice := DED.INode_TO_IDevice (itfNode := _itfParentNode);	//convert Prent Nod to Parent Device for diagnostic
				IF _itfParentDevice <> 0 THEN
					//read standard master infomation
					_itfParentDevice.GetDeviceInfo (deiInfo := _stParentInfo);
				END_IF
				_itfDevice:= DED.INode_TO_IDevice (itfNode := itfHW_Node);					//convert Node to Device for diagnostic
				IF _itfDevice <> 0 THEN
					//read standard device infomation
					_itfDevice.GetDeviceInfo (deiInfo := _stDeviceInfo);
					_pConnector := _itfDevice.Connector;
					_wType := _pConnector^.wType;
					_dwID := _pConnector^.pParameterList^.dwParameterId;
				END_IF		
				//IF Node in Level 2 and not ITFBus exist maybe it is Modbus RTU; Modbus RTU has type 91
				IF _wType = 91 THEN	
					_eBusType := DED.BUS_TYPE.MODBUS_RTU;
				//IF Node in Level 1 and not ITFBus exist maybe it is SWD 
				ELSIF _udiLoop = 1 THEN
					IF _itfDevice <> 0 THEN
						//Check Device Number if missing search for Pos in SWD tree
						_itfDevice.GetDeviceInfo (deiInfo := _stDeviceInfo);
						IF _stDeviceInfo.idInstance = 0 THEN
							_itfParentNode := itfHW_Node.ParentNode;
							_itfFirstNode := _itfParentNode.FirstChildNode;
							IF _itfFirstNode = itfHW_Node THEN
								_byModulAddress := 1;
							ELSE
								_udiSiblingNodeCount := ULINT_TO_UDINT (itfHW_Node.SiblingNodeCount);
								_itfNextNode := _itfFirstNode.NextSiblingNode;
								FOR _udiLoop := 1 TO _udiSiblingNodeCount DO			
									IF _itfNextNode = itfHW_Node THEN
										_byModulAddress := UDINT_TO_BYTE (_udiLoop +1);
										_eBusType := DED.BUS_TYPE.VEN_SPEC;	
										{IF defined (variable: _ModuleInfo)}					
										_ModuleInfo.xExecute := TRUE;
										{END_IF}
										EXIT;
									ELSE
										_itfNextNode := _itfNextNode.NextSiblingNode;	
									END_IF
								END_FOR
							END_IF
						END_IF
					END_IF			
				ELSE
					//Node in Input is not from Type Device, so something is wrong in the COnfiguration or the input is wrong
					_eBusType := DED.BUS_TYPE.UNKNOWN;
				END_IF
			ELSE
				// IF not ITF Bus and Root go to next Level
				_itfParentNode := _itfParentNode.ParentNode;
				_udiLoop := _udiLoop +1;	
			END_IF
		END_IF	
	END_WHILE
	
ELSE	 
	iErrorID := eErrorCode := teErrorCodeEaton.DeviceMissing; //wrong configuration 	
END_IF
	
xComplete := TRUE;
END_METHOD

END_FUNCTION_BLOCK

// Basic/FB/FB_BasicWithBehaviour
{attribute 'hide'}
{attribute 'reflection'}
FUNCTION_BLOCK ABSTRACT FB_BasicWithBehaviour EXTENDS FB_Basic IMPLEMENTS IBasicBehaviour, CBML.IActionProvider, CBML.IActionController
VAR_INPUT
END_VAR
VAR_OUTPUT
    // ``TRUE``: Ready condition reached
    xDone : BOOL;
    // ``TRUE``: Operation is running
    xBusy : BOOL;
    // ``TRUE``: Error condition reached
    xError : BOOL;
END_VAR
VAR	
	_iBehaviourModel 	: CBML.IBehaviourModel; 	//Interface to the Behaviour Model which will be extendet in kind Class
END_VAR

METHOD GetModelState : ERROR
VAR_INPUT
    xCommit : BOOL;
END_VAR
VAR_OUTPUT
    xDone : BOOL;
    xBusy : BOOL;
    xError : BOOL;
    xAborted : BOOL;
    iErrorID : INT;
    eState : CBML.STATE;
END_VAR
IF _iBehaviourModel <> 0 THEN
	_iBehaviourModel.GetModelState(xCommit:= xCommit, xDone=> xDone, xBusy=> xBusy, xError=> xError, xAborted=> xAborted, iErrorID=> iErrorID, eState=> eState);
END_IF
END_METHOD

(* An action controller is used whenever it is necessary to have the actions of the action controller
 instead of those of the action provider called. ``ControlCleanupAction`` is the action controller
 specifically used to control the |STATE.CLEANING| state.*)
METHOD ControlCleanupAction
VAR_INPUT
	itfCleanupActionProvider	: CBML.ICleanupActionProvider;
	xAbortProposed	: BOOL;
	iErrorIDProposed	: INT;
END_VAR
VAR_OUTPUT
	xComplete	: BOOL;
	xAbort	: BOOL;
	iErrorID	: INT;
END_VAR
CleanupAction(xAbortProposed:= xAbortProposed, iErrorIDProposed:= iErrorIDProposed, xComplete=> xComplete, xAbort=> xAbort, iErrorID=> iErrorID);
END_METHOD

(* An action controller is used whenever it is necessary to have the actions of the action controller
 instead of those of the action provider called. ``ControlCyclicAction`` is the action controller
 specifically used to control the |STATE.EXECUTING| state.*)
METHOD ControlCyclicAction
VAR_INPUT
	itfCyclicActionProvider	: CBML.ICyclicActionProvider;
	itfTimingController	: CBML.ITimingController;
END_VAR
VAR_OUTPUT
	xComplete	: BOOL;
	iErrorID	: INT;
END_VAR
CyclicAction(itfTimingController:= itfTimingController, xComplete=> xComplete, iErrorID=> iErrorID);
END_METHOD


(* Intended for releasing external resources (like RTS handles)

 Do not call other internal function block instances in the context of this method.
 Call only external functions defined inside the RTS.
 For cleaning up other resources than external ones, please use the ``CleanupAction``.
 This method should be callable in the context of ``FB_EXIT`` for example
 before downloading a new application or before reseting an application.*)
METHOD ControlExitAction
VAR_INPUT
	itfExitActionProvider	: CBML.IExitActionProvider;
	xAfterCleanup	: BOOL;
	xInCopyCode	: BOOL;
END_VAR
ExitAction(xAfterCleanup:= xAfterCleanup, xInCopyCode:= xInCopyCode);
END_METHOD


(* An action controller is used whenever it is necessary to have the actions of the action controller
 instead of those of the action provider called. ``ControlResetAction`` is the action controller
 specifically used to control the |STATE.RESETTING| state.*)
METHOD ControlResetAction
VAR_INPUT
	itfResetActionProvider	: CBML.IResetActionProvider;
END_VAR
VAR_OUTPUT
	xComplete	: BOOL;
END_VAR
ResetAction(xComplete=> xComplete);
END_METHOD


(* An action controller is used whenever it is necessary to have the actions of the action controller
 instead of those of the action provider called. ``ControlStartAction`` is the action controller
 specifically used to control the |STATE.STARTING| state.*)
METHOD ControlStartAction
VAR_INPUT
	itfStartActionProvider	: CBML.IStartActionProvider;
END_VAR
VAR_OUTPUT
	xComplete	: BOOL;
	iErrorID	: INT;
END_VAR
StartAction(xComplete=> xComplete, iErrorID=> iErrorID);
END_METHOD



METHOD CleanupAction
VAR_INPUT
    xAbortProposed : BOOL;
    iErrorIDProposed: INT;
END_VAR
VAR_OUTPUT
	{warning disable C0533}
    xComplete : BOOL := TRUE;
    xAbort: BOOL := xAbortProposed;
 	iErrorID : INT := iErrorIDProposed;
	{warning restore C0533}
END_VAR
END_METHOD

METHOD CyclicAction
VAR_INPUT
    itfTimingController : CBML.ITimingController;
END_VAR
VAR_OUTPUT
	{warning disable C0533}
    xComplete : BOOL := TRUE;
    iErrorID : INT := 0;
	{warning restore C0533}
END_VAR
END_METHOD

METHOD ExitAction
VAR_INPUT
    xAfterCleanup : BOOL;
    xInCopyCode : BOOL;
END_VAR
END_METHOD

METHOD ResetAction
VAR_OUTPUT
	{warning disable C0533}
    xComplete : BOOL := TRUE;
	{warning restore C0533}
END_VAR
END_METHOD

METHOD StartAction
VAR_OUTPUT
	{warning disable C0533}
    xComplete : BOOL := TRUE;
	iErrorID : INT := 0;
	{warning restore C0533}
END_VAR
END_METHOD

PROPERTY IBehaviourModel : CBML.IBehaviourModel
GET
IBehaviourModel:= _iBehaviourModel;
END_GET
SET
_iBehaviourModel := IBehaviourModel;
IBehaviourModel.ActionController := THIS^;
END_SET
END_PROPERTY

END_FUNCTION_BLOCK

// Basic/FB/FB_Basic
{attribute 'hide'}
{attribute 'reflection'}
{attribute 'no_assign'}
FUNCTION_BLOCK ABSTRACT FB_Basic IMPLEMENTS IBasicElement
VAR
    {attribute 'instance-path'} 
    {attribute 'noinit'}
    _strName		: STRING(255); 					// Instance path of the FB for Diagnostic
	_strOnlyName	: STRING; 						// Instance name of FB without path
	
END_VAR

//FB_Init is always available implicitly and it is used primarily for initialization.
//The return value is not evaluated. For a specific influence, you can also declare the
//methods explicitly and provide additional code there with the standard initialization
//code. You can evaluate the return value.
METHOD FB_Init: BOOL
VAR_INPUT
    bInitRetains: BOOL; // TRUE: the retain variables are initialized (reset warm / reset cold)
    bInCopyCode: BOOL;  // TRUE: the instance will be copied to the copy code afterward (online change)   
END_VAR
VAR
	_iHelpPos	: INT; //Help Variable for store Position
END_VAR
_strOnlyName := _strName;
REPEAT
_iHelpPos := Standard.FIND (STR1 := _strOnlyName, STR2:= '.');
IF _iHelpPos <> 0 THEN
	_strOnlyName := Standard.RIGHT(_strOnlyName, SIZE:= (Standard.LEN(_strOnlyName)-_iHelpPos));
END_IF

UNTIL _iHelpPos = 0
END_REPEAT
END_METHOD

//Name of instance from this FB
PROPERTY  GetName : STRING
GET
GetName := _strOnlyName;
END_GET
END_PROPERTY

//Name of instance from this FB with complete path
PROPERTY GetPath : STRING(255)
GET
GetPath := _strName;
END_GET
END_PROPERTY

END_FUNCTION_BLOCK

// Basic/Interface/IBasicElement
{attribute 'hide'}
INTERFACE IBasicElement  EXTENDS __SYSTEM.IQueryInterface

PROPERTY GetName : STRING
GET
END_GET
END_PROPERTY

PROPERTY GetPath : STRING[255]
GET
END_GET
END_PROPERTY

END_INTERFACE

// Basic/Interface/IBasicBehaviour
{attribute 'hide'}
INTERFACE IBasicBehaviour EXTENDS IBasicElement

METHOD GetModelState : ERROR
VAR_INPUT
    xCommit : BOOL;
END_VAR
VAR_OUTPUT
    xDone : BOOL;
    xBusy : BOOL;
    xError : BOOL;
    xAborted : BOOL;
    iErrorID : INT;
    eState : CBML.STATE;
END_VAR
END_METHOD

PROPERTY IBehaviourModel : CBML.IBehaviourModel
GET
END_GET
SET
END_SET
END_PROPERTY

END_INTERFACE

// Basic/Interface/I_HWDevice
{attribute 'hide'}
INTERFACE I_HWDevice EXTENDS IBasicElement

END_INTERFACE

// Interface/ITF_DIL
//Interface for a DIL SWD FB
INTERFACE ITF_DIL

//Status and Control Contactor
PROPERTY Contactor : BOOL
GET
END_GET
SET
END_SET
END_PROPERTY

//Contactor manual Switch Psoition
PROPERTY SwitchState_1_0_A : teSwitchPos_1_0_A
GET
END_GET
END_PROPERTY

END_INTERFACE

// Interface/ITF_PKE
//Interface for a PKE SWD FB
INTERFACE ITF_PKE EXTENDS ITF_Base_MotorProtection

//Acknowledge required for ZMR Function
PROPERTY ACKR : BOOL
GET
END_GET
SET
END_SET
END_PROPERTY

//Class Information from PKE, time delay
PROPERTY Class : BYTE
GET
END_GET
END_PROPERTY

//Status and Control Contactor
PROPERTY Contactor : BOOL
GET
END_GET
SET
END_SET
END_PROPERTY

//Current in A 
PROPERTY Current_A : REAL
GET
END_GET
END_PROPERTY

//Information which kind of Fieldbus is in use
PROPERTY eFieldbus : teFieldbus
GET
END_GET
END_PROPERTY

//Detail Error Code from PKE
PROPERTY ErrorCode : teErrorCodeEaton
GET
END_GET
END_PROPERTY

//Give the Current back in the defined Unit 
METHOD M_Current : REAL
VAR_INPUT
	eCurrentUnit : teCurrentUnit;	//Define the Unit of the Return Value
END_VAR
END_METHOD

//Identification Modul Name
{attribute 'analysis' := '-23'} 
PROPERTY ModulName : STRING[51]
GET
END_GET
END_PROPERTY

//Modul Present on SWD
PROPERTY ModulPresent : BOOL
GET
END_GET
END_PROPERTY

//Install Trip Block
PROPERTY PartTripBlock : teTripBlock
GET
END_GET
END_PROPERTY

//Status from PKE
PROPERTY PkeStatus : BOOL
GET
END_GET
END_PROPERTY

//Defined Max Ir Value
PROPERTY SelectValueIr : Real
GET
END_GET
END_PROPERTY

//Contactor manual Switch Psoition
PROPERTY SwitchState_1_0_A : teSwitchPos_1_0_A
GET
END_GET
END_PROPERTY

//Thermal Motor Image calculate by Motor Protection
PROPERTY ThermalMotorImage : REAL
GET
END_GET
END_PROPERTY

//Trip Reason 
PROPERTY TripReason : teTripReason
GET
END_GET
END_PROPERTY

//Set ZMR Mode to Auto or Hand
PROPERTY ZmrAutoHand : BOOL
GET
END_GET
SET
END_SET
END_PROPERTY

END_INTERFACE

// Interface/ITF_Base_MotorProtection
//Basis Information for MotorProtection Modul
INTERFACE ITF_Base_MotorProtection EXTENDS __SYSTEM.IQueryInterface

//Current in A 
PROPERTY Current_A : REAL
GET
END_GET
END_PROPERTY

// Information of Connection Status on Fieldbus
PROPERTY P_xConnected  : BOOL
GET
END_GET
END_PROPERTY

//Error happen on Device
PROPERTY P_xError : BOOL
GET
END_GET
END_PROPERTY

END_INTERFACE

// FunctionBlock/FB_Drive
//Function Block to contorl all Eaton Drives
{attribute 'conditionalshow_all_locals'}
//Function Block for handling all Eaton Drives in the same way
FUNCTION_BLOCK FB_Drive EXTENDS FB_HWDeviceBasic IMPLEMENTS ITF_Drive
VAR_INPUT
	//Commands for Drive
	stCommand			: tsCommandAndControl16bit; //Command Structure
	rSetpointSpeed		: REAL;				//Setpoint for Frequenzq Speed in Hz	
END_VAR
VAR_OUTPUT    
	//Loal Status Information from Drive                              	
	stStatus      		: tsStatusAndFaults16bit; //Status Structure 
	rActSpeed			: REAL;				//Speed in Hz
	rCurrent_A			: REAL;				//Current in A	
END_VAR
VAR
	_pstOutput : POINTER TO tsDriveCommandAndSpeed;		//Output Structure from Drive Control Word
	_pstInput	: POINTER TO tsDriveStatusAndSpeed;		//Input  Structure from Drive Status Word
	
